END_VAR
IF PR_Load THEN PR_Load_Exe(); PR_Load:=FALSE; END_IF
IF PR_Save THEN PR_Save_Exe(); PR_Save:=FALSE; END_IF
IF CA_Load THEN CA_Load_Exe(); CA_Load:=FALSE; END_IF
IF CA_Save THEN CA_Save_Exe(); CA_Save:=FALSE; END_IF
IF JL_Load THEN JL_Load_Exe(); JL_Load:=FALSE; END_IF
IF JL_Save THEN JL_Save_Exe(); JL_Save:=FALSE; END_IF
END_FUNCTION_BLOCK
ACTION CA_Load_Exe:
sFileMode:='r';
FileOpen();

IF hFile<>0 THEN

	(* Read calendar month *)
	FOR i := 0 TO 31 DO
		r1:=SysFileSetPos(File:=hFile, Pos:=(1024 + ((CA_Sel-1)*32 + i)*4));
		r2:=SysFileRead(File:=hFile, Buffer:=ADR(CA.Profile[i]), Size:=1);
	END_FOR

	(* Close file *)
	SysFileClose(File:=hFile);

	(* Validate data *)
	CA_Act :=CA_Sel;
	CN_Act :=CN_Sel;
	CN_YAct:=CN_YSel;

	Message:='Calendar load OK';

END_IF
END_ACTION
ACTION CA_Save_Exe:
sFileMode:='a';
FileOpen();

IF hFile<>0 THEN

	(* Write calendar month *)
	FOR i := 0 TO 31 DO
		r1:=SysFileSetPos(File:=hFile, Pos:=(1024 + ((CA_Sel-1)*32 + i)*4));
		r2:=SysFileGetPos(hFile);
		r2:=SysFileWrite(File:=hFile, Buffer:=ADR(CA.Profile[i]), Size:=1);
	END_FOR

	(* Close file *)
	SysFileClose(File:=hFile);

	Message:='Calendar save OK';

END_IF
END_ACTION
ACTION FileOpen:
(* Create current filename 'yyyyCRnn.DAT' *)
sFileName:=CONCAT(FilesPath,WORD_TO_STRING(CN_YSel));
sFileName:=CONCAT(STR1:=sFileName, STR2:='CR');
IF CN_Sel<10 THEN
sFileName:=CONCAT(STR1:=sFileName, STR2:='0');
END_IF
sFileName:=CONCAT(STR1:=sFileName, STR2:=BYTE_TO_STRING(CN_Sel));
sFileName:=CONCAT(STR1:=sFileName, STR2:='.DAT');

(* Check file version and size! *)
(* ... *)

(* Open data file *)
hFile:=SysFileOpen(FileName:=sFileName, Mode:='r');

(* File not found *)
IF hFile=0 THEN
	Message:='File not found - created empty file';
	(* Create empty file *)
	hFile:=SysFileOpen(FileName:=sFileName, Mode:='w');
	MEMCLR(pDestinationAddress:=ADR(Buf), BytesToClear:=SIZEOF(Buf));
	FOR i := 0 TO 10239 BY 512 DO
		SysFileWrite(File:=hFile, Buffer:=ADR(Buf), Size:=512);
	END_FOR
	Buf[0]:=1;
	SysFileSetPos(File:=hFile, Pos:=0);
	SysFileWrite(File:=hFile, Buffer:=ADR(Buf), Size:=1);
END_IF

(* Close file *)
SysFileClose(File:=hFile);

(* Open data file *)
hFile:=SysFileOpen(FileName:=sFileName, Mode:=sFileMode);
END_ACTION
ACTION JL_Load_Exe:
sFileMode:='r';
FileOpen();

IF hFile<>0 THEN

	(* Read jolly *)
	r1:=SysFileSetPos(File:=hFile, Pos:=512);
	r2:=SysFileRead(File:=hFile, Buffer:=ADR(JL), Size:=SIZEOF(JL));

	(* Close file *)
	SysFileClose(File:=hFile);

	(* Validate data *)
	CN_Act:=CN_Sel;
	CN_YAct:=CN_YSel;

	Message:='Jolly load OK';

END_IF
END_ACTION
ACTION JL_Save_Exe:
sFileMode:='a';
FileOpen();

IF hFile<>0 THEN

	(* Write selected profile *)
	r1:=SysFileSetPos(File:=hFile, Pos:=512);
	r2:=SysFileWrite(File:=hFile, Buffer:=ADR(JL), Size:=SIZEOF(JL));

	(* Close file *)
	SysFileClose(File:=hFile);

	Message:='Jolly save OK';

END_IF
END_ACTION
ACTION PR_Load_Exe:
sFileMode:='r';
FileOpen();

IF hFile<>0 THEN

	(* Read selected profile *)
	r1:=SysFileSetPos(File:=hFile, Pos:=(3072 + 512*PR_Sel));
	r2:=SysFileRead(File:=hFile, Buffer:=ADR(PR), Size:=SIZEOF(PR));

	(* Close file *)
	SysFileClose(File:=hFile);

	(* Validate data *)
	PR_Act:=PR_Sel;
	CN_Act:=CN_Sel;
	CN_YAct:=CN_YSel;

	Message:='Profile load OK';

END_IF
END_ACTION
ACTION PR_Save_Exe:
sFileMode:='a';
FileOpen();

IF hFile<>0 THEN

	(* Write selected profile *)
	r1:=SysFileSetPos(File:=hFile, Pos:=(3072 + 512*PR_Sel));
	r2:=SysFileWrite(File:=hFile, Buffer:=ADR(PR), Size:=SIZEOF(PR));

	(* Close file *)
	SysFileClose(File:=hFile);

	Message:='Profile save OK';

END_IF
END_ACTION

(* POU Plant_Objects/obj_CRONTER, ST *)
FUNCTION_BLOCK obj_CRONTER
(* === THERMOSTAT ===
   v1.0[30/07/15] - Versioning
*)
VAR_INPUT
	(* Settings *)
	ID			: BYTE;		(* Index of instanced object *)

	InitOK		: BOOL;
	Alarm		: BOOL;
	Warning		: BOOL;

	Profile		: typ_Cron_Profile; 				(* Profilo attivo *)
	ProfileNr	: BYTE;								(* Indice profilo attivo *)
	CalendarIdx : WORD;								(* Indice calendario attivo *)
	Jolly		: ARRAY[0..9] OF typ_Cron_Jolly;	(* Jolly attivi *)

	Temperature	: INT;
	Local_MaxRunTAmb	:	INT;					(* Local maximum environment temperature, NOT "TAMB" *)

	Histeresys:INT; (* isteresi per la ripartenza del Comando ON*)
END_VAR
VAR_IN_OUT
END_VAR
VAR_OUTPUT
	SetPoint		: INT;
	Run				: BOOL;
	AntifreezeForce	: BOOL;
	RunCrono		: BOOL;

	(* Status *)
	Status_Log		: BYTE;
	Status_Vis 		: DWORD;
END_VAR
VAR
	Buf: 	ARRAY[0..512] OF BYTE; (* AVOID THIS!! *)
	hFile: 	DWORD;
	sFile: 	STRING;
	sFile2: STRING;

	i:		WORD;
	t1:		DWORD;
	t2:		BOOL;

END_VAR
(* Check initialization *)
IF NOT InitOK THEN Init(); END_IF

(* Check Temperature *)
(*IF Temperature < Local_MaxRunTAmb THEN*)

	(* LOCAL environment temperature lower than maximum allowed -> Proceed with SetPoint adjustment *)
	(* Chrono *)
	IF CalendarIdx<>Sys.Time_CT_Day THEN DB_Load(); END_IF
	SetPoint:=Profile.Setpoint[Sys.Time_CT_Quarter];

	(* Check jolly *)
	FOR i := 0 TO 9 DO
		IF ( DT_TO_DWORD(Jolly[i].Start)>0  AND Jolly[i].End>Jolly[i].Start AND
		     Jolly[i].Start<=Sys.Time_CT_DT AND Jolly[i].End>Sys.Time_CT_DT ) THEN
				SetPoint:=Jolly[i].Temp;
		END_IF
	END_FOR

(*
	IF SetPoint < 180 THEN
		(* Switch off the device *)
		Run := FALSE;
	ELSE
		(* Set according to feedback T - Histeresys of 1°C *)
		IF Temperature >= (SetPoint + 5) THEN
			Run := FALSE;
		ELSIF Temperature <= (SetPoint - 5) THEN
			Run := TRUE;
		END_IF

		(* Between "SetPoint-5" and "SetPoint+5" last state (ON or OFF) of "Run" is kept	*)
	END_IF
*)

(* Gestione uscita Crono *)
		IF SetPoint>0 THEN RunCrono := TRUE;
		ELSIF SetPoint=0 THEN RunCrono := FALSE;
		END_IF

(* GEstione uscita Cronotermostato *)


		IF Temperature >= (SetPoint) THEN
			Run := FALSE;
		ELSIF Temperature <= (SetPoint - Histeresys) THEN
			Run := TRUE;
		END_IF


(*ELSE
	(* Environment overtemperature: stop heating -> Stop device *)
	Run := FALSE;
END_IF
*)
(* Freeze warning: Switch on and heat! *)
(*IF Temperature < Plant_AntiFreezeTAmb THEN AntifreezeForce := TRUE;
ELSE AntifreezeForce := FALSE;
END_IF*)



(* Status color *)
   IF Alarm   THEN Status_Log:=2; Status_Vis:=COLOR_RED;
ELSIF Warning THEN Status_Log:=1; Status_Vis:=COLOR_YELLOW;
              ELSE Status_Log:=0; Status_Vis:=COLOR_GREEN;
			  END_IF
END_FUNCTION_BLOCK
ACTION AddLogData:
Logger.s1:=INSERT('&THER=',BYTE_TO_STRING(ID),5);
IF ID<10 THEN Logger.s1:=INSERT(Logger.s1,'0',5); END_IF

Logger.s1:=CONCAT(Logger.s1,INT_TO_STRING(SetPoint));			Logger.s1:=CONCAT(Logger.s1,';');

Logger.s1:=CONCAT(Logger.s1,WORD_TO_STRING(Status_Log));
ADDSTRING(ADR(Logger.TData), ADR(Logger.s1), Logger.TLen);
END_ACTION
ACTION DB_Create:
(* Create empty file *)
hFile:=SysFileOpen(FileName:=sFile, Mode:='w');

MEMCLR(pDestinationAddress:=ADR(Buf), BytesToClear:=SIZEOF(Buf));
FOR i := 0 TO 10239 BY 512 DO
	t1:=SysFileWrite(File:=hFile, Buffer:=ADR(Buf), Size:=512);		(* Clear created file (all bytes 0) *)
END_FOR
Buf[0]:=1;
t2:=SysFileSetPos(File:=hFile, Pos:=0);
t1:=SysFileWrite(File:=hFile, Buffer:=ADR(Buf), Size:=1);
SysFileClose(File:=hFile);
END_ACTION
ACTION DB_Load:
DB_SetName();

(* Open data file *)
hFile:=SysFileOpen(FileName:=sFile, Mode:='r');

(* File not found *)
IF hFile=0 THEN
	Warning:=TRUE;
	LogEv(EL_Wrn,EO_CRON,ID,1,'No_data_file');
	DB_Create();
	(* Reopen file *)
	hFile:=SysFileOpen(FileName:=sFile, Mode:='r');
	IF hfile=0 THEN
		Alarm:=TRUE;
		LogEv(EL_Alarm,EO_CRON,ID,3,'Filesystem_error');
		RETURN;
	END_IF
END_IF

(* Check version *)
SysFileRead(File:=hFile, Buffer:=ADR(Buf), Size:=1);
IF Buf[0]<>1 THEN
	IF NOT Alarm THEN
		Alarm:=TRUE;
		LogEv(EL_Alarm,EO_CRON,ID,2,'Bad_data_version');
	END_IF
	SysFileClose(File:=hFile);
	RETURN;
END_IF

(* Read Jolly data *)
t2:=SysFileSetPos(File:=hFile, Pos:=512);
t1:=SysFileRead(File:=hFile, Buffer:=ADR(Jolly), Size:=SIZEOF(Jolly));
(* Read active profile index *)
CalendarIdx:=Sys.Time_CT_Day;
t2:=SysFileSetPos(File:=hFile, Pos:=(1024+4*CalendarIdx));
t1:=SysFileRead(File:=hFile, Buffer:=ADR(ProfileNr), Size:=SIZEOF(ProfileNr));
(* Read active profile *)
t2:=SysFileSetPos(File:=hFile, Pos:=(3072+512*ProfileNr));
t1:=SysFileRead(File:=hFile, Buffer:=ADR(Profile), Size:=SIZEOF(Profile));

(* Close file and validate data *)
SysFileClose(File:=hFile);
END_ACTION
ACTION DB_SetName:
(* Create current filename 'yyyyCRnn.DAT' *)
sFile:=CONCAT(FilesPath,WORD_TO_STRING(Sys.Time_Year));
sFile:=CONCAT(STR1:=sFile, STR2:='CR');
IF ID<10 THEN
sFile:=CONCAT(STR1:=sFile, STR2:='0');
END_IF
sFile:=CONCAT(STR1:=sFile, STR2:=BYTE_TO_STRING(ID));
sFile:=CONCAT(STR1:=sFile, STR2:='.DAT');
END_ACTION
ACTION Init:
DB_Load();
InitOK:=TRUE;
END_ACTION

(* POU Plant_Objects/obj_MODBUS_ANZFRER_01, ST *)
FUNCTION_BLOCK obj_MODBUS_ANZFRER_01
VAR CONSTANT

	TimeOutModBus: TON;


END_VAR
VAR_INPUT
	ID			:	BYTE;
	Address		:	BYTE;
	(* Modbus *)
	Refresh_Now	:	BOOL;			(* Richiesta di lettura stato macchina Immediata  *)
	retryErrMax	:	BYTE := 2;

(*	IndirizzoDaScrivere: WORD;
	DatoDaScrivere: INT;
	ScriviDato: BOOL; *)

END_VAR
VAR_IN_OUT
	ModBus		:obj_MODBUS;

END_VAR
VAR_OUTPUT
	Status_Log	:	WORD;
	Status_Vis	:	DWORD;
END_VAR
VAR

	state		:	INT;
	retry		:	BYTE;
	retryErr	:	BYTE;
	ReadTmr		:	TON := (PT:=T#5s);
	fModbusAlr:BOOL;

(*	retry_write	:	BYTE;
	fWriteStatus:	BOOL;
	fWriteMode	:	BOOL;
	fWriteReset	:	BOOL; *)

	x: INT;

	VerificaFuctionCode: INT;
	VerificaNodoLetto: INT;
	ErroreComuModBus: BOOL;
	IndiceErrore: BYTE;

	MB_BitStato: ARRAY [0..450] OF BOOL;
	MB_RegistriLetti: ARRAY [0..450] OF INT;




	AddressRead: BYTE;
	index: BYTE;
	indexErr: BYTE;


	MB_V_L1_N: DWORD;
	MB_V_L2_N: DWORD;
	MB_V_L3_N: DWORD;
	MB_V_L1_L2: DWORD;
	MB_V_L1_L3: DWORD;
	MB_V_L2_L3: DWORD;
	MB_V_IL1: DWORD;
	MB_V_IL2: DWORD;
	MB_V_IL3: DWORD;
	MB_V_F: DWORD;
	MB_V_P: DWORD;
	MB_V_Q: DWORD;
	MB_V_P_F: DWORD;
	MB_IL1_MAX: DWORD;
	MB_IL2_MAX: DWORD;
	MB_IL3_MAX: DWORD;
	MB_PF_IL1: DWORD;
	MB_PF_IL2: DWORD;
	MB_PF_IL3: DWORD;
	MB_COSPI_IL1: DWORD;
	MB_COSPI_IL2: DWORD;
	MB_COSPI_IL3: DWORD;
	MB_V_P_AVG: DWORD;
	MB_V_P_MAX: DWORD;
	MB_V_Q_MAX: DWORD;
	MB_V_Q_AVG: DWORD;
	MB_V_KWh: DWORD;
	MB_V_kVAr: DWORD;



	moreno: ARRAY [0..20] OF WORD;
END_VAR
(* Call ModBus state machine *)
Stm();


(* Seganalzione stato Frigorifero  *)
IF ErroreComuModBus OR MB_BitStato[6] OR MB_BitStato[7] THEN
		Status_Log:=2; Status_Vis:=16#2020F0;
(*	ELSIF Warning OR Warning2 THEN
		Status_Log:=1; Status_Vis:=16#20F0F0; *)
    ELSE
		Status_Log:=0;
		Status_Vis:=16#006000;
END_IF
END_FUNCTION_BLOCK
ACTION AddLogData:
Logger.s1:=INSERT('&ANZ=',BYTE_TO_STRING(ID),4);
IF ID<10 THEN Logger.s1:=INSERT(Logger.s1,'0',4); END_IF


	Logger.s1:=CONCAT(Logger.s1,(REAL_TO_STRING(DWORD_TO_REAL(MB_V_L1_N)/1000)));
	Logger.s1:=CONCAT(Logger.s1,';');
	Logger.s1:=CONCAT(Logger.s1,(REAL_TO_STRING(DWORD_TO_REAL(MB_V_L2_N)/1000)));
	Logger.s1:=CONCAT(Logger.s1,';');
	Logger.s1:=CONCAT(Logger.s1,(REAL_TO_STRING(DWORD_TO_REAL(MB_V_L3_N)/1000)));
	Logger.s1:=CONCAT(Logger.s1,';');
	Logger.s1:=CONCAT(Logger.s1,(REAL_TO_STRING(DWORD_TO_REAL(MB_V_L1_L2)/1000)));
	Logger.s1:=CONCAT(Logger.s1,';');
	Logger.s1:=CONCAT(Logger.s1,(REAL_TO_STRING(DWORD_TO_REAL(MB_V_L1_L3)/1000)));
	Logger.s1:=CONCAT(Logger.s1,';');
	Logger.s1:=CONCAT(Logger.s1,(REAL_TO_STRING(DWORD_TO_REAL(MB_V_L2_L3)/1000)));
	Logger.s1:=CONCAT(Logger.s1,';');

	Logger.s1:=CONCAT(Logger.s1,(REAL_TO_STRING(DWORD_TO_REAL(MB_V_F))));
	Logger.s1:=CONCAT(Logger.s1,';');

	Logger.s1:=CONCAT(Logger.s1,(REAL_TO_STRING(DWORD_TO_REAL(MB_V_IL1))));
	Logger.s1:=CONCAT(Logger.s1,';');
	Logger.s1:=CONCAT(Logger.s1,(REAL_TO_STRING(DWORD_TO_REAL(MB_V_IL2))));
	Logger.s1:=CONCAT(Logger.s1,';');
	Logger.s1:=CONCAT(Logger.s1,(REAL_TO_STRING(DWORD_TO_REAL(MB_V_IL3))));
	Logger.s1:=CONCAT(Logger.s1,';');

	Logger.s1:=CONCAT(Logger.s1,(REAL_TO_STRING(DWORD_TO_REAL(MB_IL1_MAX))));
	Logger.s1:=CONCAT(Logger.s1,';');
	Logger.s1:=CONCAT(Logger.s1,(REAL_TO_STRING(DWORD_TO_REAL(MB_IL1_MAX))));
	Logger.s1:=CONCAT(Logger.s1,';');
	Logger.s1:=CONCAT(Logger.s1,(REAL_TO_STRING(DWORD_TO_REAL(MB_IL1_MAX))));
	Logger.s1:=CONCAT(Logger.s1,';');


	Logger.s1:=CONCAT(Logger.s1,(REAL_TO_STRING(DWORD_TO_REAL(MB_PF_IL1))));
	Logger.s1:=CONCAT(Logger.s1,';');
	Logger.s1:=CONCAT(Logger.s1,(REAL_TO_STRING(DWORD_TO_REAL(MB_PF_IL2))));
	Logger.s1:=CONCAT(Logger.s1,';');
	Logger.s1:=CONCAT(Logger.s1,(REAL_TO_STRING(DWORD_TO_REAL(MB_PF_IL3))));
	Logger.s1:=CONCAT(Logger.s1,';');

	Logger.s1:=CONCAT(Logger.s1,(REAL_TO_STRING(DWORD_TO_REAL(MB_V_P))));
	Logger.s1:=CONCAT(Logger.s1,';');
	Logger.s1:=CONCAT(Logger.s1,(REAL_TO_STRING(DWORD_TO_REAL(MB_V_P_AVG))));
	Logger.s1:=CONCAT(Logger.s1,';');
	Logger.s1:=CONCAT(Logger.s1,(REAL_TO_STRING(DWORD_TO_REAL(MB_V_P_MAX))));
	Logger.s1:=CONCAT(Logger.s1,';');

	Logger.s1:=CONCAT(Logger.s1,(REAL_TO_STRING(DWORD_TO_REAL(MB_V_Q))));
	Logger.s1:=CONCAT(Logger.s1,';');
	Logger.s1:=CONCAT(Logger.s1,(REAL_TO_STRING(DWORD_TO_REAL(MB_V_Q_MAX))));
	Logger.s1:=CONCAT(Logger.s1,';');

	Logger.s1:=CONCAT(Logger.s1,(REAL_TO_STRING(DWORD_TO_REAL(MB_V_KWh)/100)));
	Logger.s1:=CONCAT(Logger.s1,';');
	Logger.s1:=CONCAT(Logger.s1,(REAL_TO_STRING(DWORD_TO_REAL(MB_V_kVAr)/100)));
	Logger.s1:=CONCAT(Logger.s1,';');

	Logger.s1:=CONCAT(Logger.s1,WORD_TO_STRING(Status_Log));
	Logger.s1:=CONCAT(Logger.s1,';');

	Logger.s1:=CONCAT(Logger.s1,(REAL_TO_STRING(DWORD_TO_REAL(MB_COSPI_IL1))));
	Logger.s1:=CONCAT(Logger.s1,';');
	Logger.s1:=CONCAT(Logger.s1,(REAL_TO_STRING(DWORD_TO_REAL(MB_COSPI_IL2))));
	Logger.s1:=CONCAT(Logger.s1,';');
	Logger.s1:=CONCAT(Logger.s1,(REAL_TO_STRING(DWORD_TO_REAL(MB_COSPI_IL3))));
	Logger.s1:=CONCAT(Logger.s1,';');
	Logger.s1:=CONCAT(Logger.s1,'0');    (* 0=3-phase, 1 = mono phase *)


ADDSTRING(ADR(Logger.TData), ADR(Logger.s1), Logger.TLen);
END_ACTION
ACTION Stm:
CASE state OF
	0:	(* Refresh time manager *)
		ReadTmr(IN:=NOT ReadTmr.Q);
		(*A tempo interrogo il nodo sempre che non ci sia qualcuno che lo sta interrogando in quel momento *)

		IF (ReadTmr.Q AND NodoDaInterrogareANZ=Address )OR Refresh_Now AND NOT InibiscoModbusANZ THEN
			state := 10;
			ReadTmr.PT := T#5s;
			Refresh_Now := FALSE;
			InibiscoModbusANZ := TRUE;
		END_IF

	(**** Leggo le Analogiche a Disposzione  ****)

	10:	(* richiedo lettura Holding Registere Chiller  *)

		Modbus.MB_Query.SlaveAddress := Address;
		Modbus.MB_Query.FunctionCode := 3;
		ModBus.MB_Query.Read_StartAddress := 256 ;			(* richiedo lettura altri Parametri *)
		ModBus.MB_Query.Read_Quantity := 20;
		ModBus.MB_Start := TRUE;
		state := 20;

	20:	(* Risposta all'interrogazione *)
		IF NOT ModBus.MB_Start   THEN
			VerificaFuctionCode:=ModBus.MB_Resp.FunctionCode;
			VerificaNodoLetto:=ModBus.MB_Resp.SlaveAddress;

			IF ModBus.MB_MASTER.MB_Error<>0 THEN
				state := 300;
			ELSE
				MB_V_L1_N:= ModBus.MB_Resp.Data[0]*65536 +  ModBus.MB_Resp.Data[1];   	(* Vedi tabella *)
				MB_V_L2_N:= ModBus.MB_Resp.Data[2]*65536 +  ModBus.MB_Resp.Data[3];   	(* Vedi tabella *)
				MB_V_L3_N:= ModBus.MB_Resp.Data[4]*65536 +  ModBus.MB_Resp.Data[5];   	(* Vedi tabella *)
				MB_V_L1_L2:= ModBus.MB_Resp.Data[6]*65536 +  ModBus.MB_Resp.Data[7];   	(* Vedi tabella *)
				MB_V_L1_L3:= ModBus.MB_Resp.Data[8]*65536 +  ModBus.MB_Resp.Data[9];   	(* Vedi tabella *)
				MB_V_L2_L3:= ModBus.MB_Resp.Data[10]*65536 +  ModBus.MB_Resp.Data[11];   	(* Vedi tabella *)
				ModBus.MB_Query.Read_StartAddress := 268; 	(* richiedo lettura altri Parametri *)
				ModBus.MB_Query.Read_Quantity := 10;
				ModBus.MB_Start := TRUE;

				state := 30;
			END_IF
		END_IF

	30: (* Rispota Altri paramenti *)
		IF NOT ModBus.MB_Start  THEN

			IF ModBus.MB_MASTER.MB_Error<>0 THEN
				state := 300;
			ELSE
				MB_V_IL1:= ModBus.MB_Resp.Data[0]*65536 +  ModBus.MB_Resp.Data[1];   	(* Vedi tabella *)
				MB_V_IL2:= ModBus.MB_Resp.Data[2]*65536 +  ModBus.MB_Resp.Data[3];   	(* Vedi tabella *)
				MB_V_IL3:= ModBus.MB_Resp.Data[4]*65536 +  ModBus.MB_Resp.Data[5];   	(* Vedi tabella *)
				MB_V_F:= ModBus.MB_Resp.Data[6]*65536 +  ModBus.MB_Resp.Data[7];   	(* Vedi tabella *)
				MB_V_P:= ModBus.MB_Resp.Data[8]*65536 +  ModBus.MB_Resp.Data[9];   	(* Vedi tabella *)

				ModBus.MB_Query.Read_StartAddress := 278; (* richiedo lettura altri Parametri *)
				ModBus.MB_Query.Read_Quantity := 20;
				ModBus.MB_Start := TRUE;

				state := 40;
			END_IF
		END_IF



	40: (* Rispota Altri paramenti *)
		IF NOT ModBus.MB_Start  THEN

			IF ModBus.MB_MASTER.MB_Error<>0 THEN
				state := 300;
			ELSE
				MB_V_Q:= ModBus.MB_Resp.Data[0]*65536 +  ModBus.MB_Resp.Data[1];   	(* Vedi tabella *)
				MB_V_P_F:= ModBus.MB_Resp.Data[2]*65536 +  ModBus.MB_Resp.Data[3];   	(* Vedi tabella *)
				MB_V_KWh:= ModBus.MB_Resp.Data[4]*65536 +  ModBus.MB_Resp.Data[5];   	(* Vedi tabella *)
				MB_V_kVAr:= ModBus.MB_Resp.Data[6]*65536 +  ModBus.MB_Resp.Data[7];   	(* Vedi tabella *)

				ModBus.MB_Query.Read_StartAddress := 354; (* richiedo lettura altri Parametri *)
				ModBus.MB_Query.Read_Quantity := 20;
				ModBus.MB_Start := TRUE;

				state := 50;
			END_IF
		END_IF

	50: (* Rispota Altri paramenti *)
		IF NOT ModBus.MB_Start  THEN

			IF ModBus.MB_MASTER.MB_Error<>0 THEN
				state := 300;
			ELSE

				MB_V_P_AVG:= ModBus.MB_Resp.Data[0]*65536 +  ModBus.MB_Resp.Data[1];   	(* Vedi tabella *)
				MB_V_P_MAX:= ModBus.MB_Resp.Data[2]*65536 +  ModBus.MB_Resp.Data[3];   	(* Vedi tabella *)
				MB_IL1_MAX:= ModBus.MB_Resp.Data[4]*65536 +  ModBus.MB_Resp.Data[5];   	(* Vedi tabella *)
				MB_IL2_MAX:= ModBus.MB_Resp.Data[6]*65536 +  ModBus.MB_Resp.Data[7];   	(* Vedi tabella *)
				MB_IL3_MAX:= ModBus.MB_Resp.Data[8]*65536 +  ModBus.MB_Resp.Data[9];   	(* Vedi tabella *)

				ModBus.MB_Query.Read_StartAddress := 342; (* richiedo lettura altri Parametri *)
				ModBus.MB_Query.Read_Quantity := 20;
				ModBus.MB_Start := TRUE;

				state := 55;
			END_IF
		END_IF

	55: (* Rispota Altri paramenti *)
		IF NOT ModBus.MB_Start  THEN

			IF ModBus.MB_MASTER.MB_Error<>0 THEN
				state := 300;
			ELSE
				MB_PF_IL1:= ModBus.MB_Resp.Data[0]*65536 +  ModBus.MB_Resp.Data[1];   	(* Vedi tabella *)
				MB_PF_IL2:= ModBus.MB_Resp.Data[2]*65536 +  ModBus.MB_Resp.Data[3];   	(* Vedi tabella *)
				MB_PF_IL3:= ModBus.MB_Resp.Data[4]*65536 +  ModBus.MB_Resp.Data[5];   	(* Vedi tabella *)
				MB_COSPI_IL1:= ModBus.MB_Resp.Data[6]*65536 +  ModBus.MB_Resp.Data[7];   	(* Vedi tabella *)
				MB_COSPI_IL2:= ModBus.MB_Resp.Data[8]*65536 +  ModBus.MB_Resp.Data[9];   	(* Vedi tabella *)
				MB_COSPI_IL3:= ModBus.MB_Resp.Data[10]*65536 +  ModBus.MB_Resp.Data[11];   	(* Vedi tabella *)

				ModBus.MB_Query.Read_StartAddress := 422; (* richiedo lettura altri Parametri *)
				ModBus.MB_Query.Read_Quantity := 20;
				ModBus.MB_Start := TRUE;

				state := 60;
			END_IF
		END_IF

	60: (* Rispota Altri paramenti *)
		IF NOT ModBus.MB_Start  THEN

			IF ModBus.MB_MASTER.MB_Error<>0 THEN
				state := 300;
			ELSE
				MB_V_Q_MAX:= ModBus.MB_Resp.Data[0]*65536 +  ModBus.MB_Resp.Data[1];   	(* Vedi tabella *)
				MB_V_Q_AVG:= ModBus.MB_Resp.Data[2]*65536 +  ModBus.MB_Resp.Data[3];   	(* Vedi tabella *)

				(* ModBus.MB_Query.Read_StartAddress := 422; (* richiedo lettura altri Parametri *)
				ModBus.MB_Query.Read_Quantity := 20;
				ModBus.MB_Start := TRUE; *)

				state := 295;
			END_IF
		END_IF





		295:
		IF NOT ModBus.MB_Start THEN
			IF ModBus.MB_MASTER.MB_Error<>0 THEN (*OR ModBus.MB_MASTER.MB_Error<>0 THEN*)
				state := 300;
			ELSE
				IF fModbusAlr THEN fModbusAlr := FALSE; END_IF
				NodoDaInterrogareANZ:=Address+1;
				InibiscoModbusANZ:=FALSE;
				retryErr := 0;
				retry := 0;
				state := 0;
					IF fModbusAlr=FALSE AND ErroreComuModBus=TRUE THEN
						LogEv(EL_Log,EO_CHI,ID,62,'ComunicazioneModBus_OK');
						ErroreComuModBus := FALSE;
				(*	WarningCtr := SEL(WarningCtr=0, WarningCtr-1, 0); *)
					END_IF


			END_IF
		END_IF



	(**** CHECK MODBUS ERROR ****)
	300: 	(* Release MODBUS *)
			InibiscoModbusANZ:=FALSE;
			(* Retries *)
			retry:=retry+1;
			IF retry>3 THEN
				retry:=0;

				(* Verify if slave is dead *)
				IF retryErr < retryErrMaX THEN
					retryErr := retryErr + 1;
				ELSE
					fModbusAlr := TRUE;
					(* Verify ModBus error	*)

					IF fModbusAlr AND ErroreComuModBus=FALSE THEN
						LogEv(EL_Alarm,EO_CHI,ID,61,CONCAT('ErroreModbus_',INT_TO_STRING(ModBus.MB_MASTER.MB_Error)));
						ErroreComuModBus := TRUE;
					END_IF
				END_IF

				END_IF
			Refresh_Now := FALSE;
			InibiscoModbusANZ:=FALSE;
			NodoDaInterrogareANZ:=Address+1;
			state:=0;
END_CASE




(* Controllo Time Out Ciclo ModBus *)

TimeOutModBus(In:=state<>0,PT:=t#30s);
IF TimeOutModBus.Q THEN
	State:=0;
	Refresh_Now:=TRUE;  (* Rilancio la lettura del nodo *)
	IF MODBUS.MB_Lock=TRUE THEN MODBUS.MB_Lock:=FALSE;END_IF
	IF InibiscoModbusANZ=TRUE THEN InibiscoModbusANZ:=FALSE;END_IF
END_IF
END_ACTION

(* POU Plant_Objects/obj_MODBUS_FRG_AER485P1, ST *)
FUNCTION_BLOCK obj_MODBUS_FRG_AER485P1
VAR CONSTANT

	TimeOutModBus: TON;


END_VAR
VAR_INPUT
	ID			:	BYTE;
	Address		:	BYTE;


	SetPointManuale: INT; 			(* SetPoint forazato in manuale escludendo la curva di carico *)
	AbilitaSetPointManuale : BOOL ; (* Abilita il funzionamento col set point Manaule Escludendo la curva cliamtica *)


	(* Modbus *)
	Refresh_Now	:	BOOL;			(* Richiesta di lettura stato macchina Immediata  *)
	retryErrMax	:	BYTE := 2;

	Temperatura: INT;


	STOP_REQ: BOOL;
	RUN_REQ: BOOL;
	(* Timings *)
	OnDelay		:	TIME;
	OffDelay	:	TIME;

	OnOff		: 	BOOL;

	IndirizzoDaScrivere: WORD;
	DatoDaScrivere: INT;
	ScriviDato: BOOL;

	ImpMB_2SetPoint: INT;
	ImpMB_ResetFrigo: BOOL;
	ImpMB_LocRem: BOOL;
	fWriteAttivazioneComandi:BOOL;




END_VAR
VAR_IN_OUT
	ModBus		:obj_MODBUS;
	CLIM		:typ_Clima;

END_VAR
VAR_OUTPUT
	Run			:	BOOL;

	Status_Log	:	WORD;
	Status_Vis	:	DWORD;
END_VAR
VAR
	(* da diego per gestione stato stringa > 255*)
	temp :STRING(255);
	tempRaw		: ARRAY [0..MAX_SEND_TCP_CLIENT] OF BYTE;
	tempRawLen :DINT;
	longString:STRING(800);

	(* Timer manage switch on/off delay *)
	Delay		: 	TONOF;

	AllarmeFrigo_MB		:ARRAY [0..100] OF	FLT_EVENT;
	Warning		:	FLT_TAP := (TAP:=100);

	state		:	INT;
	retry		:	BYTE;
	retryErr	:	BYTE;
	ReadTmr		:	TON := (PT:=T#5s);
	fModbusAlr:BOOL;

(*	retry_write	:	BYTE;
	fWriteStatus:	BOOL;
	fWriteMode	:	BOOL;
	fWriteReset	:	BOOL; *)

	SetPointCC: DINT;
	x: INT;
	ImpMB_SetPoint: INT;
	Ctrl_Run: BOOL;


	VerificaFuctionCode: INT;
	VerificaNodoLetto: INT;
	ErroreComuModBus: BOOL;
	IndiceErrore: BYTE;

	MB_BitStato: ARRAY [0..200] OF BOOL;
	MB_RegistriLetti: ARRAY [0..450] OF INT;


	AddressRead: BYTE;
	index: BYTE;
	indexErr: BYTE;





END_VAR
VAR_INPUT RETAIN
	ChillerAbilitato: BOOL;
END_VAR
(* Aggiornamento in tempo reale dei TON e TOFF funzionamento Pompa *)

Delay.PT_OF := OffDelay;
Delay.PT_ON := OnDelay + WORD_TO_TIME(1000*ID);

(* Check climatic setup *)
IF NOT CLIM.InitOK THEN Clima_Default(); END_IF;
(* Calculate Setpoint *)

	IF Temperatura>=CLIM.Points[0].X  THEN SetPointCC:=CLIM.Points[0].Y; END_IF;
	IF Temperatura>=CLIM.Points[1].X AND Temperatura<CLIM.Points[0].X THEN SetPointCC:=CLIM.Points[0].Y; END_IF;
	IF Temperatura>=CLIM.Points[2].X AND Temperatura<CLIM.Points[1].X THEN SetPointCC:=CLIM.Points[1].Y; END_IF;
	IF Temperatura>=CLIM.Points[3].X AND Temperatura<CLIM.Points[2].X THEN SetPointCC:=CLIM.Points[2].Y; END_IF;
	IF Temperatura>=CLIM.Points[4].X AND Temperatura<CLIM.Points[3].X THEN SetPointCC:=CLIM.Points[3].Y; END_IF;
	IF Temperatura<CLIM.Points[4].X THEN SetPointCC:=CLIM.Points[4].Y; END_IF;


	IF Temperatura<CLIM.Points[4].X THEN SetPointCC:=CLIM.Points[4].Y; END_IF;


(* Scelta del set point della cladaia o vien preso dalla curva cliamtica o da un riferimento esterno *)
IF AbilitaSetPointManuale THEN
	ImpMB_SetPoint:=(SetPointManuale);
ELSE
	ImpMB_SetPoint:=DINT_TO_INT(SetPointCC);
END_IF


(* Controllo Bit di funzionamento ON e OFF  *)
Ctrl_Run := OnOff AND ChillerAbilitato;
Delay(IN:=Ctrl_Run);



IF STOP_REQ THEN Run := 1;
	ELSIF RUN_REQ THEN Run := 0;
ELSE
	Run :=Delay.OUT AND ChillerAbilitato;
END_IF



(* Call ModBus state machine *)
Stm();

(* Check alarm	*)
CheckAlarm();



(* Seganalzione stato Frigorifero  *)
IF ErroreComuModBus OR MB_BitStato[6] OR MB_BitStato[7] THEN
		Status_Log:=2; Status_Vis:=16#2020F0;
(*	ELSIF Warning OR Warning2 THEN
		Status_Log:=1; Status_Vis:=16#20F0F0; *)
    ELSE
		Status_Log:=0;
		Status_Vis:=16#006000;
END_IF
END_FUNCTION_BLOCK
ACTION AddLogData:
Logger.s1:=INSERT('&CHI=',BYTE_TO_STRING(ID),4);
IF ID<10 THEN Logger.s1:=INSERT(Logger.s1,'0',4); END_IF

tempRawLen:=0;

temp:=Logger.s1;
ADDSTRING(ADR(tempRaw), ADR(temp), tempRawLen);

FOR x:= 1 TO 2 DO

	temp:=CONCAT(INT_TO_STRING(MB_RegistriLetti[x]),';');
	ADDSTRING(ADR(tempRaw), ADR(temp), tempRawLen);

END_FOR


FOR x:= 5 TO 15 DO
	temp:=CONCAT(INT_TO_STRING(MB_RegistriLetti[x]),';');
	ADDSTRING(ADR(tempRaw), ADR(temp), tempRawLen);
END_FOR

FOR x:= 18 TO 19 DO
	temp:=CONCAT(INT_TO_STRING(MB_RegistriLetti[x]),';');
	ADDSTRING(ADR(tempRaw), ADR(temp), tempRawLen);
END_FOR

FOR x:= 21 TO 25 DO
	temp:=CONCAT(INT_TO_STRING(MB_RegistriLetti[x]),';');
	ADDSTRING(ADR(tempRaw), ADR(temp), tempRawLen);
END_FOR

FOR x:= 180 TO 207 DO
	temp:=CONCAT(INT_TO_STRING(MB_RegistriLetti[x]),';');
	ADDSTRING(ADR(tempRaw), ADR(temp), tempRawLen);
END_FOR

FOR x:= 209 TO 232 DO
		temp:=CONCAT(INT_TO_STRING(MB_RegistriLetti[x]),';');
	ADDSTRING(ADR(tempRaw), ADR(temp), tempRawLen);
END_FOR

FOR x:= 235 TO 244 DO
	temp:=CONCAT(INT_TO_STRING(MB_RegistriLetti[x]),';');
	ADDSTRING(ADR(tempRaw), ADR(temp), tempRawLen);
END_FOR

FOR x:= 268 TO 276 DO
	temp:=CONCAT(INT_TO_STRING(MB_RegistriLetti[x]),';');
	ADDSTRING(ADR(tempRaw), ADR(temp), tempRawLen);
END_FOR

FOR x:= 408 TO 414 DO
	temp:=CONCAT(INT_TO_STRING(MB_RegistriLetti[x]),';');
	ADDSTRING(ADR(tempRaw), ADR(temp), tempRawLen);
END_FOR

FOR x:= 1 TO 19 DO
	temp:=CONCAT(SEL(MB_BitStato[x],'0','1'),';');
	ADDSTRING(ADR(tempRaw), ADR(temp), tempRawLen);
END_FOR

FOR x:= 21 TO 21 DO
	temp:=CONCAT(SEL(MB_BitStato[x],'0','1'),';');
	ADDSTRING(ADR(tempRaw), ADR(temp), tempRawLen);
END_FOR

FOR x:= 28 TO 31 DO
	temp:=CONCAT(SEL(MB_BitStato[x],'0','1'),';');
	ADDSTRING(ADR(tempRaw), ADR(temp), tempRawLen);
END_FOR

FOR x:= 34 TO 59 DO
	temp:=CONCAT(SEL(MB_BitStato[x],'0','1'),';');
	ADDSTRING(ADR(tempRaw), ADR(temp), tempRawLen);
END_FOR

FOR x:= 100 TO 198 DO
	temp:=CONCAT(SEL(MB_BitStato[x],'0','1'),';');
	ADDSTRING(ADR(tempRaw), ADR(temp), tempRawLen);
END_FOR

temp:=SEL(MB_BitStato[199],'0','1');
ADDSTRING(ADR(tempRaw), ADR(temp), tempRawLen);



(*



Logger.s1:=CONCAT(Logger.s1,(INT_TO_STRING(MB_RegistriLetti[204])); 			(* Set modo funzionamento freddo *)
Logger.s1:=CONCAT(Logger.s1,';');
Logger.s1:=CONCAT(Logger.s1,(INT_TO_STRING(MB_RegistriLetti[206]));  			(* SetCaldo Set modo funzionamento caldo *)
Logger.s1:=CONCAT(Logger.s1,';');
Logger.s1:=CONCAT(Logger.s1,WORD_TO_STRING(MB_DifGradi));  			(* Dif.Grad Set differenziale gradino per termostato *)
Logger.s1:=CONCAT(Logger.s1,';');
Logger.s1:=CONCAT(Logger.s1,WORD_TO_STRING(MB_DifTot));    			(* Dif.Tot. Set differenziale totale per termostato *)
Logger.s1:=CONCAT(Logger.s1,';');
Logger.s1:=CONCAT(Logger.s1,WORD_TO_STRING(MB_Temp_InH2O)); 		(* Temperatura ingresso acqua *)
Logger.s1:=CONCAT(Logger.s1,';');
Logger.s1:=CONCAT(Logger.s1,WORD_TO_STRING(MB_TUA_C1));				(* Temperatura uscita acqua circuito 1 *)
Logger.s1:=CONCAT(Logger.s1,';');
Logger.s1:=CONCAT(Logger.s1,WORD_TO_STRING(MB_SecondoSetFreddo));	(* Secondo set freddo *)
Logger.s1:=CONCAT(Logger.s1,';');
Logger.s1:=CONCAT(Logger.s1,WORD_TO_STRING(MB_h_CP1));				(*Ore funzionamento compressore circuito 1 *)
Logger.s1:=CONCAT(Logger.s1,';');
Logger.s1:=CONCAT(Logger.s1,WORD_TO_STRING(MB_h_CP2));				(* Ore funzionamento compressore circuito 2 *)
Logger.s1:=CONCAT(Logger.s1,';');
Logger.s1:=CONCAT(Logger.s1,WORD_TO_STRING(MB_h_CP1A));				(* Ore funzionamento compressore circuito 2 *)
Logger.s1:=CONCAT(Logger.s1,';');

Logger.s1:=CONCAT(Logger.s1,WORD_TO_STRING(Status_Log));
Logger.s1:=CONCAT(Logger.s1,';');
Logger.s1:=CONCAT(Logger.s1,SEL(ChillerAbilitato,'0','1')); (* Chiller Abilitato 0=Disabilitato   1=abilitato *)
Logger.s1:=CONCAT(Logger.s1,';');
Logger.s1:=CONCAT(Logger.s1,SEL(MB_BitStato[0],'0','1')); 	(* Comando standby/acceso (toggle)0=OFF   1=ON *)
Logger.s1:=CONCAT(Logger.s1,';');
Logger.s1:=CONCAT(Logger.s1,SEL(MB_BitStato[1],'0','1'));	(* Comando modo funzionamento freddo/caldo (toggle) 0=FREDDO 1=CALDO *)
Logger.s1:=CONCAT(Logger.s1,';');
Logger.s1:=CONCAT(Logger.s1,SEL(MB_BitStato[2],'0','1'));	(* Comando reset sicurezze1=RESET  *)
Logger.s1:=CONCAT(Logger.s1,';');
Logger.s1:=CONCAT(Logger.s1,SEL(MB_BitStato[3],'0','1'));	 (* Comando locale/remoto (toggle)0=LOCALE   1=REMOTO  *)
Logger.s1:=CONCAT(Logger.s1,';');
Logger.s1:=CONCAT(Logger.s1,SEL(MB_BitStato[6],'0','1'));	(* Stato riassunto allarmi circuito 1  *)
Logger.s1:=CONCAT(Logger.s1,';');
Logger.s1:=CONCAT(Logger.s1,SEL(MB_BitStato[7],'0','1'));	(* Stato riassunto allarmi circuito 2  *)
Logger.s1:=CONCAT(Logger.s1,';');
Logger.s1:=CONCAT(Logger.s1,SEL(MB_BitStato[8],'0','1'));	(* Allarme flussostato *)
Logger.s1:=CONCAT(Logger.s1,';');
Logger.s1:=CONCAT(Logger.s1,SEL(MB_BitStato[12],'0','1'));	(*  Allarme termica compressore circuito 1  *)
Logger.s1:=CONCAT(Logger.s1,';');
Logger.s1:=CONCAT(Logger.s1,SEL(MB_BitStato[13],'0','1'));	(*  Allarme bassa pressione circuito 1   *)
Logger.s1:=CONCAT(Logger.s1,';');
Logger.s1:=CONCAT(Logger.s1,SEL(MB_BitStato[14],'0','1'));	(*  Allarme alta pressione circuito 1   *)
Logger.s1:=CONCAT(Logger.s1,';');
Logger.s1:=CONCAT(Logger.s1,SEL(MB_BitStato[15],'0','1'));	(*   Allarme antigelo circuito 1   *)
Logger.s1:=CONCAT(Logger.s1,';');
Logger.s1:=CONCAT(Logger.s1,SEL(MB_BitStato[16],'0','1'));	(*    Allarme termica ventilatore circuito 1   *)
Logger.s1:=CONCAT(Logger.s1,';');
Logger.s1:=CONCAT(Logger.s1,SEL(MB_BitStato[19],'0','1'));	(*  Allarme termica compressore circuito 2  *)
Logger.s1:=CONCAT(Logger.s1,';');
Logger.s1:=CONCAT(Logger.s1,SEL(MB_BitStato[20],'0','1'));  (*  Allarme bassa pressione circuito 2   *)
Logger.s1:=CONCAT(Logger.s1,';');
Logger.s1:=CONCAT(Logger.s1,SEL(MB_BitStato[21],'0','1'));  (*  Allarme alta pressione circuito 2   *)
Logger.s1:=CONCAT(Logger.s1,';');
Logger.s1:=CONCAT(Logger.s1,SEL(MB_BitStato[22],'0','1'));  (*   Allarme antigelo circuito 2   *)
Logger.s1:=CONCAT(Logger.s1,';');
Logger.s1:=CONCAT(Logger.s1,SEL(MB_BitStato[23],'0','1'));  (*    Allarme termica ventilatore circuito 2   *)
Logger.s1:=CONCAT(Logger.s1,';');
Logger.s1:=CONCAT(Logger.s1,SEL(MB_BitStato[26],'0','1'));  (*    Allarme monitore di tensione   *)
Logger.s1:=CONCAT(Logger.s1,';');
Logger.s1:=CONCAT(Logger.s1,SEL(MB_BitStato[29],'0','1'));  (*    Allarme Eprom   *)
Logger.s1:=CONCAT(Logger.s1,';');
Logger.s1:=CONCAT(Logger.s1,SEL(MB_BitStato[31],'0','1'));  (*     Carico pompa evaporatore   *)
Logger.s1:=CONCAT(Logger.s1,';');
Logger.s1:=CONCAT(Logger.s1,SEL(MB_BitStato[34],'0','1'));  (*      Carico compressore circuito 1   *)
Logger.s1:=CONCAT(Logger.s1,';');
Logger.s1:=CONCAT(Logger.s1,SEL(MB_BitStato[38],'0','1'));  (*       Carico ventilatore circuito 1   *)
Logger.s1:=CONCAT(Logger.s1,';');
Logger.s1:=CONCAT(Logger.s1,SEL(MB_BitStato[40],'0','1'));  (*        Carico valvola liquido circuito 1   *)
Logger.s1:=CONCAT(Logger.s1,';');
Logger.s1:=CONCAT(Logger.s1,SEL(MB_BitStato[41],'0','1'));  (*         Carico compressore secondario circuito 1   *)
Logger.s1:=CONCAT(Logger.s1,';');
Logger.s1:=CONCAT(Logger.s1,SEL(MB_BitStato[42],'0','1'));  (*         Carico compressore circuito 2   *)
Logger.s1:=CONCAT(Logger.s1,';');
Logger.s1:=CONCAT(Logger.s1,SEL(MB_BitStato[46],'0','1'));  (*         Carico ventilatore circuito 2    *)
Logger.s1:=CONCAT(Logger.s1,';');
Logger.s1:=CONCAT(Logger.s1,SEL(MB_BitStato[48],'0','1'));  (*          Carico valvola liquido circuito 2    *)
Logger.s1:=CONCAT(Logger.s1,';');
Logger.s1:=CONCAT(Logger.s1,SEL(MB_BitStato[81],'0','1'));  (*           Allarme termica compressore circuito 1A     *)
Logger.s1:=CONCAT(Logger.s1,';');
Logger.s1:=CONCAT(Logger.s1,SEL(MB_BitStato[86],'0','1'));  (*          Allarme antigelo evaporatore circuito 1     *)
Logger.s1:=CONCAT(Logger.s1,';');
Logger.s1:=CONCAT(Logger.s1,SEL(MB_BitStato[87],'0','1'));  (*          Allarme antigelo evaporatore circuito 2     *)




*)


ADDSTRING(ADR(Logger.TData), ADR(tempRaw), Logger.TLen);
END_ACTION
ACTION CheckAlarm:
(**** GEstione Log ad Evento *****)


FOR x:=0 TO 100 DO

	AllarmeFrigo_MB[x](IN:=MB_BitStato[x+100] );

	IF AllarmeFrigo_MB[x].EVH THEN
		LogEv(EL_Log,EO_CHI,ID,x+100,CONCAT ('Allarme Attivo n. ', INT_TO_STRING(x+100)));
	END_IF

	IF AllarmeFrigo_MB[x].EVL THEN
		LogEv(EL_Log,EO_CHI,ID,x+100,CONCAT ('Allarme Rientrato n. ', INT_TO_STRING(x+100)));
	END_IF

END_FOR
END_ACTION
ACTION Clima_Default:
IF CLIM.Points[0].X=0 THEN
	CLIM.Points[0].X:=-300; CLIM.Points[0].Y:=770;
	CLIM.Points[1].X:=-70 ; CLIM.Points[1].Y:=770;
	CLIM.Points[2].X:= 80; 	CLIM.Points[2].Y:=690;
	CLIM.Points[3].X:= 200; CLIM.Points[3].Y:=300;
	CLIM.Points[4].X:= 500; CLIM.Points[4].Y:=200;
END_IF
CLIM.InitOK:=TRUE;
LogEv(EL_Wrn,EO_chi,ID,0,'Climatic_default');
END_ACTION
ACTION Stm:
CASE state OF
	0:	(* Refresh time manager *)
		ReadTmr(IN:=NOT ReadTmr.Q);
		(*A tempo interrogo il nodo sempre che non ci sia qualcuno che lo sta interrogando in quel momento *)

		IF (ReadTmr.Q AND NodoDaInterrogareChiller=Address )OR Refresh_Now AND NOT InibiscoModbusChiller THEN
			state := 10;
			ReadTmr.PT := T#5s;  (* moreno *)
			Refresh_Now := FALSE;
			InibiscoModbusChiller := TRUE;
		END_IF

	(**** Leggo le Analogiche a Disposzione  ****)

	10:	(* richiedo lettura Holding Registere Chiller  *)

		Modbus.MB_Query.SlaveAddress := Address;
		Modbus.MB_Query.FunctionCode := 3;
		ModBus.MB_Query.Read_StartAddress := 0 ;			(* richiedo lettura altri Parametri *)
		ModBus.MB_Query.Read_Quantity := 3;
		ModBus.MB_Start := TRUE;
		state := 20;

	20:	(* Risposta all'interrogazione *)
		IF NOT ModBus.MB_Start   THEN
			VerificaFuctionCode:=ModBus.MB_Resp.FunctionCode;
			VerificaNodoLetto:=ModBus.MB_Resp.SlaveAddress;

			IF ModBus.MB_MASTER.MB_Error<>0 THEN
				state := 300;
			ELSE
				MB_RegistriLetti[0] := ModBus.MB_Resp.Data[0];   	(* Vedi tabella *)
				MB_RegistriLetti[1] := ModBus.MB_Resp.Data[1];		(* Vedi tabella *)
				MB_RegistriLetti[2] := ModBus.MB_Resp.Data[2];		(* Vedi tabella *)


				ModBus.MB_Query.Read_StartAddress := 5; 	(* richiedo lettura altri Parametri *)
				ModBus.MB_Query.Read_Quantity := 11;
				ModBus.MB_Start := TRUE;

				state := 30;
			END_IF
		END_IF

	30: (* Rispota Altri paramenti *)
		IF NOT ModBus.MB_Start  THEN

			IF ModBus.MB_MASTER.MB_Error<>0 THEN
				state := 300;
			ELSE
				MB_RegistriLetti[5] := ModBus.MB_Resp.Data[0];   	(* Vedi tabella *)
				MB_RegistriLetti[6] := ModBus.MB_Resp.Data[1];		(* Vedi tabella *)
				MB_RegistriLetti[7] := ModBus.MB_Resp.Data[2];		(* Vedi tabella *)
				MB_RegistriLetti[8] := ModBus.MB_Resp.Data[3];		(* Vedi tabella *)
				MB_RegistriLetti[9] := ModBus.MB_Resp.Data[4];		(* Vedi tabella *)
				MB_RegistriLetti[10] := ModBus.MB_Resp.Data[5];		(* Vedi tabella *)
				MB_RegistriLetti[11] := ModBus.MB_Resp.Data[6];		(* Vedi tabella *)
				MB_RegistriLetti[12] := ModBus.MB_Resp.Data[7];		(* Vedi tabella *)
				MB_RegistriLetti[13] := ModBus.MB_Resp.Data[8];		(* Vedi tabella *)
				MB_RegistriLetti[14] := ModBus.MB_Resp.Data[9];		(* Vedi tabella *)
				MB_RegistriLetti[15] := ModBus.MB_Resp.Data[10];		(* Vedi tabella *)

				ModBus.MB_Query.Read_StartAddress := 21; (* richiedo lettura altri Parametri *)
				ModBus.MB_Query.Read_Quantity := 5;
				ModBus.MB_Start := TRUE;

				state := 40;
			END_IF
		END_IF

	40: (* Rispota Altri paramenti *)
		IF NOT ModBus.MB_Start  THEN

			IF ModBus.MB_MASTER.MB_Error<>0 THEN
				state := 300;
			ELSE
				MB_RegistriLetti[21] := ModBus.MB_Resp.Data[0];   	(* Vedi tabella *)
				MB_RegistriLetti[22] := ModBus.MB_Resp.Data[1];		(* Vedi tabella *)
				MB_RegistriLetti[23] := ModBus.MB_Resp.Data[2];		(* Vedi tabella *)
				MB_RegistriLetti[24] := ModBus.MB_Resp.Data[3];		(* Vedi tabella *)
				MB_RegistriLetti[25] := ModBus.MB_Resp.Data[4];		(* Vedi tabella *)

				ModBus.MB_Query.Read_StartAddress := 180; (* richiedo lettura altri Parametri *)
				ModBus.MB_Query.Read_Quantity := 20;
				ModBus.MB_Start := TRUE;

				state := 45;
			END_IF
		END_IF

	45: (* Rispota Altri paramenti *)
		IF NOT ModBus.MB_Start  THEN

			IF ModBus.MB_MASTER.MB_Error<>0 THEN
				state := 300;
			ELSE
				MB_RegistriLetti[180] := ModBus.MB_Resp.Data[0];   	(* Vedi tabella *)
				MB_RegistriLetti[181] := ModBus.MB_Resp.Data[1];		(* Vedi tabella *)
				MB_RegistriLetti[182] := ModBus.MB_Resp.Data[2];		(* Vedi tabella *)
				MB_RegistriLetti[183] := ModBus.MB_Resp.Data[3];		(* Vedi tabella *)
				MB_RegistriLetti[184] := ModBus.MB_Resp.Data[4];		(* Vedi tabella *)
				MB_RegistriLetti[185] := ModBus.MB_Resp.Data[5];		(* Vedi tabella *)
				MB_RegistriLetti[186] := ModBus.MB_Resp.Data[6];		(* Vedi tabella *)
				MB_RegistriLetti[187] := ModBus.MB_Resp.Data[7];		(* Vedi tabella *)
				MB_RegistriLetti[188] := ModBus.MB_Resp.Data[8];		(* Vedi tabella *)
				MB_RegistriLetti[189] := ModBus.MB_Resp.Data[9];		(* Vedi tabella *)
				MB_RegistriLetti[190] := ModBus.MB_Resp.Data[10];		(* Vedi tabella *)
				MB_RegistriLetti[191] := ModBus.MB_Resp.Data[11];		(* Vedi tabella *)
				MB_RegistriLetti[192] := ModBus.MB_Resp.Data[12];		(* Vedi tabella *)
				MB_RegistriLetti[193] := ModBus.MB_Resp.Data[13];		(* Vedi tabella *)
				MB_RegistriLetti[194] := ModBus.MB_Resp.Data[14];		(* Vedi tabella *)
				MB_RegistriLetti[195] := ModBus.MB_Resp.Data[15];		(* Vedi tabella *)
				MB_RegistriLetti[196] := ModBus.MB_Resp.Data[16];		(* Vedi tabella *)
				MB_RegistriLetti[197] := ModBus.MB_Resp.Data[17];		(* Vedi tabella *)
				MB_RegistriLetti[198] := ModBus.MB_Resp.Data[18];		(* Vedi tabella *)
				MB_RegistriLetti[199] := ModBus.MB_Resp.Data[19];		(* Vedi tabella *)

				ModBus.MB_Query.Read_StartAddress := 200; (* richiedo lettura altri Parametri *)
				ModBus.MB_Query.Read_Quantity := 9;
				ModBus.MB_Start := TRUE;

				state := 50;
			END_IF
		END_IF
	50: (* Rispota Altri paramenti *)
		IF NOT ModBus.MB_Start  THEN

			IF ModBus.MB_MASTER.MB_Error<>0 THEN
				state := 300;
			ELSE
				MB_RegistriLetti[200] := ModBus.MB_Resp.Data[0];   	(* Vedi tabella *)
				MB_RegistriLetti[201] := ModBus.MB_Resp.Data[1];		(* Vedi tabella *)
				MB_RegistriLetti[202] := ModBus.MB_Resp.Data[2];		(* Vedi tabella *)
				MB_RegistriLetti[203] := ModBus.MB_Resp.Data[3];		(* Vedi tabella *)
				MB_RegistriLetti[204] := ModBus.MB_Resp.Data[4];		(* Vedi tabella *)
				MB_RegistriLetti[205] := ModBus.MB_Resp.Data[5];		(* Vedi tabella *)
				MB_RegistriLetti[206] := ModBus.MB_Resp.Data[6];		(* Vedi tabella *)
				MB_RegistriLetti[207] := ModBus.MB_Resp.Data[7];		(* Vedi tabella *)

				ModBus.MB_Query.Read_StartAddress := 209; (* richiedo lettura altri Parametri *)
				ModBus.MB_Query.Read_Quantity := 20;
				ModBus.MB_Start := TRUE;

				state := 55;
			END_IF
		END_IF

	55: (* Rispota Altri paramenti *)
		IF NOT ModBus.MB_Start  THEN

			IF ModBus.MB_MASTER.MB_Error<>0 THEN
				state := 300;
			ELSE
				MB_RegistriLetti[209] := ModBus.MB_Resp.Data[0];   	(* Vedi tabella *)
				MB_RegistriLetti[210] := ModBus.MB_Resp.Data[1];		(* Vedi tabella *)
				MB_RegistriLetti[211] := ModBus.MB_Resp.Data[2];		(* Vedi tabella *)
				MB_RegistriLetti[212] := ModBus.MB_Resp.Data[3];		(* Vedi tabella *)
				MB_RegistriLetti[213] := ModBus.MB_Resp.Data[4];		(* Vedi tabella *)
				MB_RegistriLetti[214] := ModBus.MB_Resp.Data[5];		(* Vedi tabella *)
				MB_RegistriLetti[215] := ModBus.MB_Resp.Data[6];		(* Vedi tabella *)
				MB_RegistriLetti[216] := ModBus.MB_Resp.Data[7];		(* Vedi tabella *)
				MB_RegistriLetti[217] := ModBus.MB_Resp.Data[8];		(* Vedi tabella *)
				MB_RegistriLetti[218] := ModBus.MB_Resp.Data[9];		(* Vedi tabella *)
				MB_RegistriLetti[219] := ModBus.MB_Resp.Data[10];		(* Vedi tabella *)
				MB_RegistriLetti[220] := ModBus.MB_Resp.Data[11];		(* Vedi tabella *)
				MB_RegistriLetti[221] := ModBus.MB_Resp.Data[12];		(* Vedi tabella *)
				MB_RegistriLetti[222] := ModBus.MB_Resp.Data[13];		(* Vedi tabella *)
				MB_RegistriLetti[223] := ModBus.MB_Resp.Data[14];		(* Vedi tabella *)
				MB_RegistriLetti[224] := ModBus.MB_Resp.Data[15];		(* Vedi tabella *)
				MB_RegistriLetti[225] := ModBus.MB_Resp.Data[16];		(* Vedi tabella *)
				MB_RegistriLetti[226] := ModBus.MB_Resp.Data[17];		(* Vedi tabella *)
				MB_RegistriLetti[227] := ModBus.MB_Resp.Data[18];		(* Vedi tabella *)
				MB_RegistriLetti[228] := ModBus.MB_Resp.Data[19];		(* Vedi tabella *)

				ModBus.MB_Query.Read_StartAddress := 229; (* richiedo lettura altri Parametri *)
				ModBus.MB_Query.Read_Quantity := 4;
				ModBus.MB_Start := TRUE;

				state := 60;
			END_IF
		END_IF

	60: (* Rispota Altri paramenti *)
		IF NOT ModBus.MB_Start  THEN

			IF ModBus.MB_MASTER.MB_Error<>0 THEN
				state := 300;
			ELSE
				MB_RegistriLetti[229] := ModBus.MB_Resp.Data[0];   	(* Vedi tabella *)
				MB_RegistriLetti[230] := ModBus.MB_Resp.Data[1];		(* Vedi tabella *)
				MB_RegistriLetti[231] := ModBus.MB_Resp.Data[2];		(* Vedi tabella *)
				MB_RegistriLetti[232] := ModBus.MB_Resp.Data[3];		(* Vedi tabella *)

				ModBus.MB_Query.Read_StartAddress := 235; (* richiedo lettura altri Parametri *)
				ModBus.MB_Query.Read_Quantity := 10;
				ModBus.MB_Start := TRUE;

				state := 65;
			END_IF
		END_IF


	65: (* Rispota Altri paramenti *)
		IF NOT ModBus.MB_Start  THEN

			IF ModBus.MB_MASTER.MB_Error<>0 THEN
				state := 300;
			ELSE
				MB_RegistriLetti[235] := ModBus.MB_Resp.Data[0];   	(* Vedi tabella *)
				MB_RegistriLetti[236] := ModBus.MB_Resp.Data[1];		(* Vedi tabella *)
				MB_RegistriLetti[237] := ModBus.MB_Resp.Data[2];		(* Vedi tabella *)
				MB_RegistriLetti[238] := ModBus.MB_Resp.Data[3];		(* Vedi tabella *)
				MB_RegistriLetti[239] := ModBus.MB_Resp.Data[4];		(* Vedi tabella *)
				MB_RegistriLetti[240] := ModBus.MB_Resp.Data[5];		(* Vedi tabella *)
				MB_RegistriLetti[241] := ModBus.MB_Resp.Data[6];		(* Vedi tabella *)
				MB_RegistriLetti[242] := ModBus.MB_Resp.Data[7];		(* Vedi tabella *)
				MB_RegistriLetti[243] := ModBus.MB_Resp.Data[8];		(* Vedi tabella *)
				MB_RegistriLetti[244] := ModBus.MB_Resp.Data[9];		(* Vedi tabella *)

				ModBus.MB_Query.Read_StartAddress := 268; (* richiedo lettura altri Parametri *)
				ModBus.MB_Query.Read_Quantity := 9;
				ModBus.MB_Start := TRUE;

				state := 70;
			END_IF
		END_IF

	70: (* Rispota Altri paramenti *)
		IF NOT ModBus.MB_Start  THEN

			IF ModBus.MB_MASTER.MB_Error<>0 THEN
				state := 300;
			ELSE
				MB_RegistriLetti[235] := ModBus.MB_Resp.Data[0];   	(* Vedi tabella *)
				MB_RegistriLetti[236] := ModBus.MB_Resp.Data[1];		(* Vedi tabella *)
				MB_RegistriLetti[237] := ModBus.MB_Resp.Data[2];		(* Vedi tabella *)
				MB_RegistriLetti[238] := ModBus.MB_Resp.Data[3];		(* Vedi tabella *)
				MB_RegistriLetti[239] := ModBus.MB_Resp.Data[4];		(* Vedi tabella *)
				MB_RegistriLetti[240] := ModBus.MB_Resp.Data[5];		(* Vedi tabella *)
				MB_RegistriLetti[241] := ModBus.MB_Resp.Data[6];		(* Vedi tabella *)
				MB_RegistriLetti[242] := ModBus.MB_Resp.Data[7];		(* Vedi tabella *)
				MB_RegistriLetti[243] := ModBus.MB_Resp.Data[8];		(* Vedi tabella *)
				MB_RegistriLetti[244] := ModBus.MB_Resp.Data[9];		(* Vedi tabella *)

				ModBus.MB_Query.Read_StartAddress := 268; (* richiedo lettura altri Parametri *)
				ModBus.MB_Query.Read_Quantity := 9;
				ModBus.MB_Start := TRUE;

				state := 75;
			END_IF
		END_IF


	75: (* Rispota Altri paramenti *)
		IF NOT ModBus.MB_Start  THEN

			IF ModBus.MB_MASTER.MB_Error<>0 THEN
				state := 300;
			ELSE
				MB_RegistriLetti[268] := ModBus.MB_Resp.Data[0];   	(* Vedi tabella *)
				MB_RegistriLetti[269] := ModBus.MB_Resp.Data[1];		(* Vedi tabella *)
				MB_RegistriLetti[270] := ModBus.MB_Resp.Data[2];		(* Vedi tabella *)
				MB_RegistriLetti[271] := ModBus.MB_Resp.Data[3];		(* Vedi tabella *)
				MB_RegistriLetti[272] := ModBus.MB_Resp.Data[4];		(* Vedi tabella *)
				MB_RegistriLetti[273] := ModBus.MB_Resp.Data[5];		(* Vedi tabella *)
				MB_RegistriLetti[274] := ModBus.MB_Resp.Data[6];		(* Vedi tabella *)
				MB_RegistriLetti[275] := ModBus.MB_Resp.Data[7];		(* Vedi tabella *)
				MB_RegistriLetti[276] := ModBus.MB_Resp.Data[8];		(* Vedi tabella *)

				ModBus.MB_Query.Read_StartAddress := 408; (* richiedo lettura altri Parametri *)
				ModBus.MB_Query.Read_Quantity := 6;
				ModBus.MB_Start := TRUE;

				state := 80;
			END_IF
		END_IF

	80: (* Rispota Altri paramenti *)
		IF NOT ModBus.MB_Start  THEN

			IF ModBus.MB_MASTER.MB_Error<>0 THEN
				state := 300;
			ELSE
				MB_RegistriLetti[408] := ModBus.MB_Resp.Data[0];   		(* Vedi tabella *)
				MB_RegistriLetti[409] := ModBus.MB_Resp.Data[1];		(* Vedi tabella *)
				MB_RegistriLetti[410] := ModBus.MB_Resp.Data[2];		(* Vedi tabella *)
				MB_RegistriLetti[411] := ModBus.MB_Resp.Data[3];		(* Vedi tabella *)
				MB_RegistriLetti[412] := ModBus.MB_Resp.Data[4];		(* Vedi tabella *)
				MB_RegistriLetti[413] := ModBus.MB_Resp.Data[5];		(* Vedi tabella *)

				ModBus.MB_Query.Read_StartAddress := 408; (* richiedo lettura altri Parametri *)
				ModBus.MB_Query.Read_Quantity := 6;
				ModBus.MB_Start := TRUE;

				state := 100;
			END_IF
		END_IF






	100: (* Rispota Altri paramenti COIL *)
		IF NOT ModBus.MB_Start  THEN

			IF ModBus.MB_MASTER.MB_Error<>0 THEN
				state := 300;
			ELSE
				Modbus.MB_Query.SlaveAddress := Address;
				Modbus.MB_Query.FunctionCode := 1;
				ModBus.MB_Query.Read_StartAddress := 0;	(* richiedo lettura altri Parametri *)
				ModBus.MB_Query.Read_Quantity := 60;
				ModBus.MB_Start := TRUE;

				state:=105;
			END_IF
		END_IF
	105: (* Rispota Altri paramenti *)

		IF NOT ModBus.MB_Start  THEN

			IF ModBus.MB_MASTER.MB_Error<>0 THEN
				state := 300;
			ELSE

				MB_BitStato[1]:=ModBus.MB_MASTER.ReceiveBuffer.Data[3].0; (*Vedi Tabella *)
				MB_BitStato[2]:=ModBus.MB_MASTER.ReceiveBuffer.Data[3].1; (*Vedi Tabella *)
				MB_BitStato[3]:=ModBus.MB_MASTER.ReceiveBuffer.Data[3].2; (*Vedi Tabella *)
				MB_BitStato[4]:=ModBus.MB_MASTER.ReceiveBuffer.Data[3].3; (*Vedi Tabella *)
				MB_BitStato[5]:=ModBus.MB_MASTER.ReceiveBuffer.Data[3].4; (*Vedi Tabella *)
				MB_BitStato[6]:=ModBus.MB_MASTER.ReceiveBuffer.Data[3].5; (*Vedi Tabella *)
				MB_BitStato[7]:=ModBus.MB_MASTER.ReceiveBuffer.Data[3].6; (*Vedi Tabella *)
				MB_BitStato[8]:=ModBus.MB_MASTER.ReceiveBuffer.Data[3].7; (*Vedi Tabella *)
				MB_BitStato[9]:=ModBus.MB_MASTER.ReceiveBuffer.Data[4].0; (*Vedi Tabella *)
				MB_BitStato[10]:=ModBus.MB_MASTER.ReceiveBuffer.Data[4].1; (*Vedi Tabella *)
				MB_BitStato[11]:=ModBus.MB_MASTER.ReceiveBuffer.Data[4].2; (*Vedi Tabella *)
				MB_BitStato[12]:=ModBus.MB_MASTER.ReceiveBuffer.Data[4].3; (*Vedi Tabella *)
				MB_BitStato[13]:=ModBus.MB_MASTER.ReceiveBuffer.Data[4].4; (*Vedi Tabella *)
				MB_BitStato[14]:=ModBus.MB_MASTER.ReceiveBuffer.Data[4].5; (*Vedi Tabella *)
				MB_BitStato[15]:=ModBus.MB_MASTER.ReceiveBuffer.Data[4].6; (*Vedi Tabella *)
				MB_BitStato[16]:=ModBus.MB_MASTER.ReceiveBuffer.Data[4].7; (*Vedi Tabella *)
				MB_BitStato[17]:=ModBus.MB_MASTER.ReceiveBuffer.Data[5].0; (*Vedi Tabella *)
				MB_BitStato[18]:=ModBus.MB_MASTER.ReceiveBuffer.Data[5].1; (*Vedi Tabella *)
				MB_BitStato[19]:=ModBus.MB_MASTER.ReceiveBuffer.Data[5].2; (*Vedi Tabella *)
				MB_BitStato[20]:=ModBus.MB_MASTER.ReceiveBuffer.Data[5].3; (*Vedi Tabella *)
				MB_BitStato[21]:=ModBus.MB_MASTER.ReceiveBuffer.Data[5].4; (*Vedi Tabella *)
				MB_BitStato[22]:=ModBus.MB_MASTER.ReceiveBuffer.Data[5].5; (*Vedi Tabella *)
				MB_BitStato[23]:=ModBus.MB_MASTER.ReceiveBuffer.Data[5].6; (*Vedi Tabella *)
				MB_BitStato[24]:=ModBus.MB_MASTER.ReceiveBuffer.Data[5].7; (*Vedi Tabella *)
				MB_BitStato[25]:=ModBus.MB_MASTER.ReceiveBuffer.Data[6].0; (*Vedi Tabella *)
				MB_BitStato[26]:=ModBus.MB_MASTER.ReceiveBuffer.Data[6].1; (*Vedi Tabella *)
				MB_BitStato[27]:=ModBus.MB_MASTER.ReceiveBuffer.Data[6].2; (*Vedi Tabella *)
				MB_BitStato[28]:=ModBus.MB_MASTER.ReceiveBuffer.Data[6].3; (*Vedi Tabella *)
				MB_BitStato[29]:=ModBus.MB_MASTER.ReceiveBuffer.Data[6].4; (*Vedi Tabella *)
				MB_BitStato[30]:=ModBus.MB_MASTER.ReceiveBuffer.Data[6].5; (*Vedi Tabella *)
				MB_BitStato[31]:=ModBus.MB_MASTER.ReceiveBuffer.Data[6].6; (*Vedi Tabella *)
				MB_BitStato[32]:=ModBus.MB_MASTER.ReceiveBuffer.Data[6].7; (*Vedi Tabella *)
				MB_BitStato[33]:=ModBus.MB_MASTER.ReceiveBuffer.Data[7].0; (*Vedi Tabella *)
				MB_BitStato[34]:=ModBus.MB_MASTER.ReceiveBuffer.Data[7].1; (*Vedi Tabella *)
				MB_BitStato[35]:=ModBus.MB_MASTER.ReceiveBuffer.Data[7].2; (*Vedi Tabella *)
				MB_BitStato[36]:=ModBus.MB_MASTER.ReceiveBuffer.Data[7].3; (*Vedi Tabella *)
				MB_BitStato[37]:=ModBus.MB_MASTER.ReceiveBuffer.Data[7].4; (*Vedi Tabella *)
				MB_BitStato[38]:=ModBus.MB_MASTER.ReceiveBuffer.Data[7].5; (*Vedi Tabella *)
				MB_BitStato[39]:=ModBus.MB_MASTER.ReceiveBuffer.Data[7].6; (*Vedi Tabella *)
				MB_BitStato[40]:=ModBus.MB_MASTER.ReceiveBuffer.Data[7].7; (*Vedi Tabella *)
				MB_BitStato[41]:=ModBus.MB_MASTER.ReceiveBuffer.Data[8].0; (*Vedi Tabella *)
				MB_BitStato[42]:=ModBus.MB_MASTER.ReceiveBuffer.Data[8].1; (*Vedi Tabella *)
				MB_BitStato[43]:=ModBus.MB_MASTER.ReceiveBuffer.Data[8].2; (*Vedi Tabella *)
				MB_BitStato[44]:=ModBus.MB_MASTER.ReceiveBuffer.Data[8].3; (*Vedi Tabella *)
				MB_BitStato[45]:=ModBus.MB_MASTER.ReceiveBuffer.Data[8].4; (*Vedi Tabella *)
				MB_BitStato[46]:=ModBus.MB_MASTER.ReceiveBuffer.Data[8].5; (*Vedi Tabella *)
				MB_BitStato[47]:=ModBus.MB_MASTER.ReceiveBuffer.Data[8].6; (*Vedi Tabella *)
				MB_BitStato[48]:=ModBus.MB_MASTER.ReceiveBuffer.Data[8].7; (*Vedi Tabella *)
				MB_BitStato[49]:=ModBus.MB_MASTER.ReceiveBuffer.Data[9].0; (*Vedi Tabella *)
				MB_BitStato[50]:=ModBus.MB_MASTER.ReceiveBuffer.Data[9].1; (*Vedi Tabella *)
				MB_BitStato[51]:=ModBus.MB_MASTER.ReceiveBuffer.Data[9].2; (*Vedi Tabella *)
				MB_BitStato[52]:=ModBus.MB_MASTER.ReceiveBuffer.Data[9].3; (*Vedi Tabella *)
				MB_BitStato[53]:=ModBus.MB_MASTER.ReceiveBuffer.Data[9].4; (*Vedi Tabella *)
				MB_BitStato[54]:=ModBus.MB_MASTER.ReceiveBuffer.Data[9].5; (*Vedi Tabella *)
				MB_BitStato[55]:=ModBus.MB_MASTER.ReceiveBuffer.Data[9].6; (*Vedi Tabella *)
				MB_BitStato[56]:=ModBus.MB_MASTER.ReceiveBuffer.Data[9].7; (*Vedi Tabella *)
				MB_BitStato[57]:=ModBus.MB_MASTER.ReceiveBuffer.Data[10].0; (*Vedi Tabella *)
				MB_BitStato[58]:=ModBus.MB_MASTER.ReceiveBuffer.Data[10].1; (*Vedi Tabella *)
				MB_BitStato[59]:=ModBus.MB_MASTER.ReceiveBuffer.Data[10].2; (*Vedi Tabella *)
				MB_BitStato[60]:=ModBus.MB_MASTER.ReceiveBuffer.Data[10].3; (*Vedi Tabella *)
				MB_BitStato[61]:=ModBus.MB_MASTER.ReceiveBuffer.Data[10].4; (*Vedi Tabella *)
				MB_BitStato[62]:=ModBus.MB_MASTER.ReceiveBuffer.Data[10].5; (*Vedi Tabella *)
				MB_BitStato[63]:=ModBus.MB_MASTER.ReceiveBuffer.Data[10].6; (*Vedi Tabella *)
				MB_BitStato[64]:=ModBus.MB_MASTER.ReceiveBuffer.Data[10].7; (*Vedi Tabella *)


				state:=110;

			END_IF
		END_IF


	110: (* Rispota Altri paramenti *)
		IF NOT ModBus.MB_Start  THEN

			IF ModBus.MB_MASTER.MB_Error<>0 THEN
				state := 300;
			ELSE
				Modbus.MB_Query.SlaveAddress := Address;
				Modbus.MB_Query.FunctionCode := 1;
				ModBus.MB_Query.Read_StartAddress := 100;
				ModBus.MB_Query.Read_Quantity := 100;
				ModBus.MB_Start := TRUE;

				state:=115;
			END_IF
		END_IF
	115: (* Rispota Altri paramenti *)

		IF NOT ModBus.MB_Start  THEN

			IF ModBus.MB_MASTER.MB_Error<>0 THEN
				state := 300;
			ELSE

				MB_BitStato[100]:=ModBus.MB_MASTER.ReceiveBuffer.Data[3].0; (*Vedi Tabella *)
				MB_BitStato[101]:=ModBus.MB_MASTER.ReceiveBuffer.Data[3].1; (*Vedi Tabella *)
				MB_BitStato[102]:=ModBus.MB_MASTER.ReceiveBuffer.Data[3].2; (*Vedi Tabella *)
				MB_BitStato[103]:=ModBus.MB_MASTER.ReceiveBuffer.Data[3].3; (*Vedi Tabella *)
				MB_BitStato[104]:=ModBus.MB_MASTER.ReceiveBuffer.Data[3].4; (*Vedi Tabella *)
				MB_BitStato[105]:=ModBus.MB_MASTER.ReceiveBuffer.Data[3].5; (*Vedi Tabella *)
				MB_BitStato[106]:=ModBus.MB_MASTER.ReceiveBuffer.Data[3].6; (*Vedi Tabella *)
				MB_BitStato[107]:=ModBus.MB_MASTER.ReceiveBuffer.Data[3].7; (*Vedi Tabella *)
				MB_BitStato[108]:=ModBus.MB_MASTER.ReceiveBuffer.Data[4].0; (*Vedi Tabella *)
				MB_BitStato[109]:=ModBus.MB_MASTER.ReceiveBuffer.Data[4].1; (*Vedi Tabella *)
				MB_BitStato[110]:=ModBus.MB_MASTER.ReceiveBuffer.Data[4].2; (*Vedi Tabella *)
				MB_BitStato[111]:=ModBus.MB_MASTER.ReceiveBuffer.Data[4].3; (*Vedi Tabella *)
				MB_BitStato[112]:=ModBus.MB_MASTER.ReceiveBuffer.Data[4].4; (*Vedi Tabella *)
				MB_BitStato[113]:=ModBus.MB_MASTER.ReceiveBuffer.Data[4].5; (*Vedi Tabella *)
				MB_BitStato[114]:=ModBus.MB_MASTER.ReceiveBuffer.Data[4].6; (*Vedi Tabella *)
				MB_BitStato[115]:=ModBus.MB_MASTER.ReceiveBuffer.Data[4].7; (*Vedi Tabella *)
				MB_BitStato[116]:=ModBus.MB_MASTER.ReceiveBuffer.Data[5].0; (*Vedi Tabella *)
				MB_BitStato[117]:=ModBus.MB_MASTER.ReceiveBuffer.Data[5].1; (*Vedi Tabella *)
				MB_BitStato[118]:=ModBus.MB_MASTER.ReceiveBuffer.Data[5].2; (*Vedi Tabella *)
				MB_BitStato[119]:=ModBus.MB_MASTER.ReceiveBuffer.Data[5].3; (*Vedi Tabella *)
				MB_BitStato[120]:=ModBus.MB_MASTER.ReceiveBuffer.Data[5].4; (*Vedi Tabella *)
				MB_BitStato[121]:=ModBus.MB_MASTER.ReceiveBuffer.Data[5].5; (*Vedi Tabella *)
				MB_BitStato[122]:=ModBus.MB_MASTER.ReceiveBuffer.Data[5].6; (*Vedi Tabella *)
				MB_BitStato[123]:=ModBus.MB_MASTER.ReceiveBuffer.Data[5].7; (*Vedi Tabella *)
				MB_BitStato[124]:=ModBus.MB_MASTER.ReceiveBuffer.Data[6].0; (*Vedi Tabella *)
				MB_BitStato[125]:=ModBus.MB_MASTER.ReceiveBuffer.Data[6].1; (*Vedi Tabella *)
				MB_BitStato[126]:=ModBus.MB_MASTER.ReceiveBuffer.Data[6].2; (*Vedi Tabella *)
				MB_BitStato[127]:=ModBus.MB_MASTER.ReceiveBuffer.Data[6].3; (*Vedi Tabella *)
				MB_BitStato[128]:=ModBus.MB_MASTER.ReceiveBuffer.Data[6].4; (*Vedi Tabella *)
				MB_BitStato[129]:=ModBus.MB_MASTER.ReceiveBuffer.Data[6].5; (*Vedi Tabella *)
				MB_BitStato[130]:=ModBus.MB_MASTER.ReceiveBuffer.Data[6].6; (*Vedi Tabella *)
				MB_BitStato[131]:=ModBus.MB_MASTER.ReceiveBuffer.Data[6].7; (*Vedi Tabella *)
				MB_BitStato[132]:=ModBus.MB_MASTER.ReceiveBuffer.Data[7].0; (*Vedi Tabella *)
				MB_BitStato[133]:=ModBus.MB_MASTER.ReceiveBuffer.Data[7].1; (*Vedi Tabella *)
				MB_BitStato[134]:=ModBus.MB_MASTER.ReceiveBuffer.Data[7].2; (*Vedi Tabella *)
				MB_BitStato[135]:=ModBus.MB_MASTER.ReceiveBuffer.Data[7].3; (*Vedi Tabella *)
				MB_BitStato[136]:=ModBus.MB_MASTER.ReceiveBuffer.Data[7].4; (*Vedi Tabella *)
				MB_BitStato[137]:=ModBus.MB_MASTER.ReceiveBuffer.Data[7].5; (*Vedi Tabella *)
				MB_BitStato[138]:=ModBus.MB_MASTER.ReceiveBuffer.Data[7].6; (*Vedi Tabella *)
				MB_BitStato[139]:=ModBus.MB_MASTER.ReceiveBuffer.Data[7].7; (*Vedi Tabella *)
				MB_BitStato[140]:=ModBus.MB_MASTER.ReceiveBuffer.Data[8].0; (*Vedi Tabella *)
				MB_BitStato[141]:=ModBus.MB_MASTER.ReceiveBuffer.Data[8].1; (*Vedi Tabella *)
				MB_BitStato[142]:=ModBus.MB_MASTER.ReceiveBuffer.Data[8].2; (*Vedi Tabella *)
				MB_BitStato[143]:=ModBus.MB_MASTER.ReceiveBuffer.Data[8].3; (*Vedi Tabella *)
				MB_BitStato[144]:=ModBus.MB_MASTER.ReceiveBuffer.Data[8].4; (*Vedi Tabella *)
				MB_BitStato[145]:=ModBus.MB_MASTER.ReceiveBuffer.Data[8].5; (*Vedi Tabella *)
				MB_BitStato[146]:=ModBus.MB_MASTER.ReceiveBuffer.Data[8].6; (*Vedi Tabella *)
				MB_BitStato[147]:=ModBus.MB_MASTER.ReceiveBuffer.Data[8].7; (*Vedi Tabella *)
				MB_BitStato[148]:=ModBus.MB_MASTER.ReceiveBuffer.Data[9].0; (*Vedi Tabella *)
				MB_BitStato[149]:=ModBus.MB_MASTER.ReceiveBuffer.Data[9].1; (*Vedi Tabella *)
				MB_BitStato[150]:=ModBus.MB_MASTER.ReceiveBuffer.Data[9].2; (*Vedi Tabella *)
				MB_BitStato[151]:=ModBus.MB_MASTER.ReceiveBuffer.Data[9].3; (*Vedi Tabella *)
				MB_BitStato[152]:=ModBus.MB_MASTER.ReceiveBuffer.Data[9].4; (*Vedi Tabella *)
				MB_BitStato[153]:=ModBus.MB_MASTER.ReceiveBuffer.Data[9].5; (*Vedi Tabella *)
				MB_BitStato[154]:=ModBus.MB_MASTER.ReceiveBuffer.Data[9].6; (*Vedi Tabella *)
				MB_BitStato[155]:=ModBus.MB_MASTER.ReceiveBuffer.Data[9].7; (*Vedi Tabella *)
				MB_BitStato[156]:=ModBus.MB_MASTER.ReceiveBuffer.Data[10].0; (*Vedi Tabella *)
				MB_BitStato[157]:=ModBus.MB_MASTER.ReceiveBuffer.Data[10].1; (*Vedi Tabella *)
				MB_BitStato[158]:=ModBus.MB_MASTER.ReceiveBuffer.Data[10].2; (*Vedi Tabella *)
				MB_BitStato[159]:=ModBus.MB_MASTER.ReceiveBuffer.Data[10].3; (*Vedi Tabella *)
				MB_BitStato[160]:=ModBus.MB_MASTER.ReceiveBuffer.Data[10].4; (*Vedi Tabella *)
				MB_BitStato[161]:=ModBus.MB_MASTER.ReceiveBuffer.Data[10].5; (*Vedi Tabella *)
				MB_BitStato[162]:=ModBus.MB_MASTER.ReceiveBuffer.Data[10].6; (*Vedi Tabella *)
				MB_BitStato[163]:=ModBus.MB_MASTER.ReceiveBuffer.Data[10].7; (*Vedi Tabella *)
				MB_BitStato[164]:=ModBus.MB_MASTER.ReceiveBuffer.Data[11].0; (*Vedi Tabella *)
				MB_BitStato[165]:=ModBus.MB_MASTER.ReceiveBuffer.Data[11].1; (*Vedi Tabella *)
				MB_BitStato[166]:=ModBus.MB_MASTER.ReceiveBuffer.Data[11].2; (*Vedi Tabella *)
				MB_BitStato[167]:=ModBus.MB_MASTER.ReceiveBuffer.Data[11].3; (*Vedi Tabella *)
				MB_BitStato[168]:=ModBus.MB_MASTER.ReceiveBuffer.Data[11].4; (*Vedi Tabella *)
				MB_BitStato[169]:=ModBus.MB_MASTER.ReceiveBuffer.Data[11].5; (*Vedi Tabella *)
				MB_BitStato[170]:=ModBus.MB_MASTER.ReceiveBuffer.Data[11].6; (*Vedi Tabella *)
				MB_BitStato[171]:=ModBus.MB_MASTER.ReceiveBuffer.Data[11].7; (*Vedi Tabella *)
				MB_BitStato[172]:=ModBus.MB_MASTER.ReceiveBuffer.Data[12].0; (*Vedi Tabella *)
				MB_BitStato[173]:=ModBus.MB_MASTER.ReceiveBuffer.Data[12].1; (*Vedi Tabella *)
				MB_BitStato[174]:=ModBus.MB_MASTER.ReceiveBuffer.Data[12].2; (*Vedi Tabella *)
				MB_BitStato[175]:=ModBus.MB_MASTER.ReceiveBuffer.Data[12].3; (*Vedi Tabella *)
				MB_BitStato[176]:=ModBus.MB_MASTER.ReceiveBuffer.Data[12].4; (*Vedi Tabella *)
				MB_BitStato[177]:=ModBus.MB_MASTER.ReceiveBuffer.Data[12].5; (*Vedi Tabella *)
				MB_BitStato[178]:=ModBus.MB_MASTER.ReceiveBuffer.Data[12].6; (*Vedi Tabella *)
				MB_BitStato[179]:=ModBus.MB_MASTER.ReceiveBuffer.Data[12].7; (*Vedi Tabella *)
				MB_BitStato[180]:=ModBus.MB_MASTER.ReceiveBuffer.Data[13].0; (*Vedi Tabella *)
				MB_BitStato[181]:=ModBus.MB_MASTER.ReceiveBuffer.Data[13].1; (*Vedi Tabella *)
				MB_BitStato[182]:=ModBus.MB_MASTER.ReceiveBuffer.Data[13].2; (*Vedi Tabella *)
				MB_BitStato[183]:=ModBus.MB_MASTER.ReceiveBuffer.Data[13].3; (*Vedi Tabella *)
				MB_BitStato[184]:=ModBus.MB_MASTER.ReceiveBuffer.Data[13].4; (*Vedi Tabella *)
				MB_BitStato[185]:=ModBus.MB_MASTER.ReceiveBuffer.Data[13].5; (*Vedi Tabella *)
				MB_BitStato[186]:=ModBus.MB_MASTER.ReceiveBuffer.Data[13].6; (*Vedi Tabella *)
				MB_BitStato[187]:=ModBus.MB_MASTER.ReceiveBuffer.Data[13].7; (*Vedi Tabella *)
				MB_BitStato[188]:=ModBus.MB_MASTER.ReceiveBuffer.Data[13].0; (*Vedi Tabella *)
				MB_BitStato[189]:=ModBus.MB_MASTER.ReceiveBuffer.Data[13].1; (*Vedi Tabella *)
				MB_BitStato[190]:=ModBus.MB_MASTER.ReceiveBuffer.Data[13].2; (*Vedi Tabella *)
				MB_BitStato[191]:=ModBus.MB_MASTER.ReceiveBuffer.Data[13].3; (*Vedi Tabella *)
				MB_BitStato[192]:=ModBus.MB_MASTER.ReceiveBuffer.Data[13].4; (*Vedi Tabella *)
				MB_BitStato[193]:=ModBus.MB_MASTER.ReceiveBuffer.Data[13].5; (*Vedi Tabella *)
				MB_BitStato[194]:=ModBus.MB_MASTER.ReceiveBuffer.Data[13].6; (*Vedi Tabella *)
				MB_BitStato[195]:=ModBus.MB_MASTER.ReceiveBuffer.Data[13].7; (*Vedi Tabella *)
				MB_BitStato[196]:=ModBus.MB_MASTER.ReceiveBuffer.Data[14].0; (*Vedi Tabella *)
				MB_BitStato[197]:=ModBus.MB_MASTER.ReceiveBuffer.Data[14].1; (*Vedi Tabella *)
				MB_BitStato[198]:=ModBus.MB_MASTER.ReceiveBuffer.Data[14].2; (*Vedi Tabella *)
				MB_BitStato[199]:=ModBus.MB_MASTER.ReceiveBuffer.Data[14].3; (*Vedi Tabella *)


				state:=200;

			END_IF
		END_IF


	200:
		IF NOT ModBus.MB_Start  THEN

			IF ModBus.MB_MASTER.MB_Error<>0 THEN
				state := 300;
			ELSE
				IF ScriviDato THEN
					state := 205;
				ELSE
					state := 295;
				END_IF
			END_IF
		END_IF


	 205:	(* Scrivo la Variabile all'indirizzo specificato  *)

		Modbus.MB_Query.SlaveAddress := Address;
		Modbus.MB_Query.FunctionCode := 6;
		ModBus.MB_Query.Write_StartAddress := IndirizzoDaScrivere;
		ModBus.MB_Query.Write_Quantity :=1;
		ModBus.MB_Query.Write_Data[0] := DatoDaScrivere;
		ModBus.MB_Start := TRUE;

		state := 295;



		295:
		IF NOT ModBus.MB_Start THEN
			IF ModBus.MB_MASTER.MB_Error<>0 THEN (*OR ModBus.MB_MASTER.MB_Error<>0 THEN*)
				state := 300;
			ELSE
				IF fModbusAlr THEN fModbusAlr := FALSE; END_IF
				NodoDaInterrogareChiller:=Address+1;
				InibiscoModbusChiller:=FALSE;
				retryErr := 0;
				retry := 0;
				state := 0;
					IF fModbusAlr=FALSE AND ErroreComuModBus=TRUE THEN
						LogEv(EL_Log,EO_CHI,ID,62,'ComunicazioneModBus_OK');
						ErroreComuModBus := FALSE;
				(*	WarningCtr := SEL(WarningCtr=0, WarningCtr-1, 0); *)
					END_IF


			END_IF
		END_IF



	(**** CHECK MODBUS ERROR ****)
	300: 	(* Release MODBUS *)
			InibiscoModbusChiller:=FALSE;
			(* Retries *)
			retry:=retry+1;
			IF retry>3 THEN
				retry:=0;

				(* Verify if slave is dead *)
				IF retryErr < retryErrMaX THEN
					retryErr := retryErr + 1;
				ELSE
					fModbusAlr := TRUE;
					(* Verify ModBus error	*)

					IF fModbusAlr AND ErroreComuModBus=FALSE THEN
						LogEv(EL_Alarm,EO_CHI,ID,61,CONCAT('ErroreModbus_',INT_TO_STRING(ModBus.MB_MASTER.MB_Error)));
						ErroreComuModBus := TRUE;
					END_IF
				END_IF

				END_IF
			Refresh_Now := FALSE;
			NodoDaInterrogareChiller:=Address+1;
			state:=0;
END_CASE




(* Controllo Time Out Ciclo ModBus *)

TimeOutModBus(In:=state<>0,PT:=t#30s);
IF TimeOutModBus.Q THEN
	State:=0;
	Refresh_Now:=TRUE;  (* Rilancio la lettura del nodo *)
	IF MODBUS.MB_Lock=TRUE THEN MODBUS.MB_Lock:=FALSE;END_IF
	IF InibiscoModbusChiller=TRUE THEN InibiscoModbusChiller:=FALSE;END_IF
END_IF
END_ACTION

(* POU Utils Functions/TONOF, ST *)
FUNCTION_BLOCK TONOF
VAR_INPUT
	IN		: BOOL;
	PT_ON	: TIME; (* time to pass, before OUT is set *)
	PT_OF	: TIME; (* time to pass, before OUT is reset *)
END_VAR
VAR_OUTPUT
	OUT		: BOOL;
END_VAR
VAR
	timer	: TON;
END_VAR
IF IN<>OUT THEN
	timer(IN:=TRUE,PT:=SEL(IN,PT_OF,PT_ON));
	IF timer.Q THEN OUT:=IN; END_IF
ELSE
	timer(IN:=FALSE);
END_IF
END_FUNCTION_BLOCK

(* POU Plant_Objects/obj_MODBUS_TRENDCOIN_01, ST *)
FUNCTION_BLOCK obj_MODBUS_TRENDCOIN_01
VAR CONSTANT

	TimeOutModBus: TON;


END_VAR
VAR_INPUT
	ID			:	BYTE;
	Address		:	BYTE;
	(* Modbus *)
	Refresh_Now	:	BOOL;			(* Richiesta di lettura stato macchina Immediata  *)
	retryErrMax	:	BYTE := 2;

(*	IndirizzoDaScrivere: WORD;
	DatoDaScrivere: INT;
	ScriviDato: BOOL; *)

END_VAR
VAR_IN_OUT
	ModBus		:obj_MODBUS;

END_VAR
VAR_OUTPUT
	Status_Log	:	WORD;
	Status_Vis	:	DWORD;
END_VAR
VAR

	state		:	INT;
	retry		:	BYTE;
	retryErr	:	BYTE;
	ReadTmr		:	TON := (PT:=T#5s);
	fModbusAlr:BOOL;

(*	retry_write	:	BYTE;
	fWriteStatus:	BOOL;
	fWriteMode	:	BOOL;
	fWriteReset	:	BOOL; *)

	x: INT;

	VerificaFuctionCode: INT;
	VerificaNodoLetto: INT;
	ErroreComuModBus: BOOL;
	IndiceErrore: BYTE;

	MB_BitStato: ARRAY [0..450] OF BOOL;
	MB_RegistriLetti: ARRAY [0..450] OF INT;

	MB_RegistriHoldingLetti: ARRAY [0..170] OF INT;
	MB_BitStatoCoil: ARRAY [0..100] OF BOOL;



	AddressRead: BYTE;
	index: BYTE;
	indexErr: BYTE;


	MB_V_L1_N: DWORD;
	MB_V_L2_N: DWORD;
	MB_V_L3_N: DWORD;
	MB_V_L1_L2: DWORD;
	MB_V_L1_L3: DWORD;
	MB_V_IL1: DWORD;
	MB_V_IL2: DWORD;
	MB_V_IL3: DWORD;
	MB_V_F: DWORD;
	MB_V_P: DWORD;
	MB_V_Q: DWORD;
	MB_V_P_F: DWORD;



	Read_StartAddress: INT;
	Read_Quantity: BYTE;
	IndiceMBLettura: INT;
	IndiceMBLetto: INT;
	test_Address: INT;
	Test_ScriviCoil: BOOL;
	test_Write: WORD;
	ScriviMB: BOOL;
END_VAR
(* Call ModBus state machine *)
Stm();

(* Check alarm	*)




(* Seganalzione stato Frigorifero  *)
IF ErroreComuModBus THEN
		Status_Log:=2; Status_Vis:=16#2020F0;
(*	ELSIF Warning OR Warning2 THEN
		Status_Log:=1; Status_Vis:=16#20F0F0; *)
    ELSE
		Status_Log:=0;
		Status_Vis:=16#006000;
END_IF
END_FUNCTION_BLOCK
ACTION AddLogData:
Logger.s1:=INSERT('&UTA=',BYTE_TO_STRING(ID),4);
IF ID<10 THEN Logger.s1:=INSERT(Logger.s1,'0',4); END_IF
(*

	Logger.s1:=CONCAT(Logger.s1,DWORD_TO_STRING(MB_V_L1_N));
	Logger.s1:=CONCAT(Logger.s1,';');
	Logger.s1:=CONCAT(Logger.s1,DWORD_TO_STRING(MB_V_L2_N));
	Logger.s1:=CONCAT(Logger.s1,';');
	Logger.s1:=CONCAT(Logger.s1,DWORD_TO_STRING(MB_V_L3_N));
	Logger.s1:=CONCAT(Logger.s1,';');
	Logger.s1:=CONCAT(Logger.s1,DWORD_TO_STRING(MB_V_L1_L2));
	Logger.s1:=CONCAT(Logger.s1,';');
	Logger.s1:=CONCAT(Logger.s1,DWORD_TO_STRING(MB_V_L1_L3));
	Logger.s1:=CONCAT(Logger.s1,';');
	Logger.s1:=CONCAT(Logger.s1,DWORD_TO_STRING(MB_V_IL1));
	Logger.s1:=CONCAT(Logger.s1,';');
	Logger.s1:=CONCAT(Logger.s1,DWORD_TO_STRING(MB_V_IL2));
	Logger.s1:=CONCAT(Logger.s1,';');
	Logger.s1:=CONCAT(Logger.s1,DWORD_TO_STRING(MB_V_IL3));
	Logger.s1:=CONCAT(Logger.s1,';');
	Logger.s1:=CONCAT(Logger.s1,DWORD_TO_STRING(MB_V_F));
	Logger.s1:=CONCAT(Logger.s1,';');
	Logger.s1:=CONCAT(Logger.s1,DWORD_TO_STRING(MB_V_P));
	Logger.s1:=CONCAT(Logger.s1,';');
	Logger.s1:=CONCAT(Logger.s1,DWORD_TO_STRING(MB_V_Q));
	Logger.s1:=CONCAT(Logger.s1,';');
	Logger.s1:=CONCAT(Logger.s1,DWORD_TO_STRING(MB_V_P_F));
*)


ADDSTRING(ADR(Logger.TData), ADR(Logger.s1), Logger.TLen);
END_ACTION
ACTION Stm:
CASE state OF
	0:	(* Refresh time manager *)
		ReadTmr(IN:=NOT ReadTmr.Q);
		(*A tempo interrogo il nodo sempre che non ci sia qualcuno che lo sta interrogando in quel momento *)

		IF (ReadTmr.Q AND NodoDaInterrogareMB1=Address )OR Refresh_Now AND NOT InibiscoModbusMB1 THEN
			state := 10;
			ReadTmr.PT := T#10s;  (* moreno *)
			Refresh_Now := FALSE;
			InibiscoModbusMB1 := TRUE;
		END_IF

	(**** Leggo le Analogiche a Disposzione  ****)

	10:	(* richiedo lettura di tutti gli Input Register   *)

		Modbus.MB_Query.SlaveAddress := Address;
		Modbus.MB_Query.FunctionCode := 4;
		Read_StartAddress := 0 ;			(* richiedo lettura altri Parametri *)
		Read_Quantity := 20;
		ModBus.MB_Start := TRUE;
		state := 20;


	20:
		ModBus.MB_Query.Read_StartAddress := 0 ;			(* richiedo lettura altri Parametri *)
		ModBus.MB_Query.Read_Quantity := 20;
		ModBus.MB_Start := TRUE;
		Read_StartAddress := 0 ;
		state := 30;



	30:	(* Risposta all'interrogazione *)
		IF NOT ModBus.MB_Start   THEN
			VerificaFuctionCode:=ModBus.MB_Resp.FunctionCode;
			VerificaNodoLetto:=ModBus.MB_Resp.SlaveAddress;

			IF ModBus.MB_MASTER.MB_Error<>0 THEN
				state := 300;
			ELSE

				FOR x:= 0 TO ModBus.MB_Query.Read_Quantity DO
					MB_RegistriLetti[Read_StartAddress+x ] := ModBus.MB_Resp.Data[x];   	(* Vedi tabella *)
				END_FOR

			ModBus.MB_Query.Read_StartAddress := 20 ;			(* richiedo lettura altri Parametri *)
			ModBus.MB_Query.Read_Quantity := 20;
			ModBus.MB_Start := TRUE;
			Read_StartAddress := 20 ;
			state := 31;
			END_IF
		END_IF


	31:	(* Risposta all'interrogazione *)
		IF NOT ModBus.MB_Start   THEN
			VerificaFuctionCode:=ModBus.MB_Resp.FunctionCode;
			VerificaNodoLetto:=ModBus.MB_Resp.SlaveAddress;

			IF ModBus.MB_MASTER.MB_Error<>0 THEN
				state := 300;
			ELSE

				FOR x:= 0 TO ModBus.MB_Query.Read_Quantity DO
					MB_RegistriLetti[Read_StartAddress+x ] := ModBus.MB_Resp.Data[x];   	(* Vedi tabella *)
				END_FOR

			ModBus.MB_Query.Read_StartAddress := 40 ;			(* richiedo lettura altri Parametri *)
			ModBus.MB_Query.Read_Quantity := 20;
			ModBus.MB_Start := TRUE;
			Read_StartAddress := 40 ;
			state := 32;
			END_IF
		END_IF



	32:	(* Risposta all'interrogazione *)
		IF NOT ModBus.MB_Start   THEN
			VerificaFuctionCode:=ModBus.MB_Resp.FunctionCode;
			VerificaNodoLetto:=ModBus.MB_Resp.SlaveAddress;

			IF ModBus.MB_MASTER.MB_Error<>0 THEN
				state := 300;
			ELSE

				FOR x:= 0 TO ModBus.MB_Query.Read_Quantity DO
					MB_RegistriLetti[Read_StartAddress+x ] := ModBus.MB_Resp.Data[x];   	(* Vedi tabella *)
				END_FOR

			ModBus.MB_Query.Read_StartAddress := 60 ;			(* richiedo lettura altri Parametri *)
			ModBus.MB_Query.Read_Quantity := 20;
			ModBus.MB_Start := TRUE;
			Read_StartAddress := 60 ;
			state := 33;
			END_IF
		END_IF

	33:	(* Risposta all'interrogazione *)
		IF NOT ModBus.MB_Start   THEN
			VerificaFuctionCode:=ModBus.MB_Resp.FunctionCode;
			VerificaNodoLetto:=ModBus.MB_Resp.SlaveAddress;

			IF ModBus.MB_MASTER.MB_Error<>0 THEN
				state := 300;
			ELSE

				FOR x:= 0 TO ModBus.MB_Query.Read_Quantity DO
					MB_RegistriLetti[Read_StartAddress+x ] := ModBus.MB_Resp.Data[x];   	(* Vedi tabella *)
				END_FOR

			ModBus.MB_Query.Read_StartAddress := 80 ;			(* richiedo lettura altri Parametri *)
			ModBus.MB_Query.Read_Quantity := 20;
			ModBus.MB_Start := TRUE;
			Read_StartAddress := 80 ;
			state := 34;
			END_IF
		END_IF


	34:	(* Risposta all'interrogazione *)
		IF NOT ModBus.MB_Start   THEN
			VerificaFuctionCode:=ModBus.MB_Resp.FunctionCode;
			VerificaNodoLetto:=ModBus.MB_Resp.SlaveAddress;

			IF ModBus.MB_MASTER.MB_Error<>0 THEN
				state := 300;
			ELSE

				FOR x:= 0 TO ModBus.MB_Query.Read_Quantity DO
					MB_RegistriLetti[Read_StartAddress+x ] := ModBus.MB_Resp.Data[x];   	(* Vedi tabella *)
				END_FOR

			ModBus.MB_Query.Read_StartAddress := 100 ;			(* richiedo lettura altri Parametri *)
			ModBus.MB_Query.Read_Quantity := 20;
			ModBus.MB_Start := TRUE;
			Read_StartAddress := 100 ;
			state := 35;
			END_IF
		END_IF


	35:	(* Risposta all'interrogazione *)
		IF NOT ModBus.MB_Start   THEN
			VerificaFuctionCode:=ModBus.MB_Resp.FunctionCode;
			VerificaNodoLetto:=ModBus.MB_Resp.SlaveAddress;

			IF ModBus.MB_MASTER.MB_Error<>0 THEN
				state := 300;
			ELSE

				FOR x:= 0 TO ModBus.MB_Query.Read_Quantity DO
					MB_RegistriLetti[Read_StartAddress+x ] := ModBus.MB_Resp.Data[x];   	(* Vedi tabella *)
				END_FOR

			ModBus.MB_Query.Read_StartAddress := 120 ;			(* richiedo lettura altri Parametri *)
			ModBus.MB_Query.Read_Quantity := 20;
			ModBus.MB_Start := TRUE;
			Read_StartAddress := 120 ;
			state := 36;
			END_IF
		END_IF

	36:	(* Risposta all'interrogazione *)
		IF NOT ModBus.MB_Start   THEN
			VerificaFuctionCode:=ModBus.MB_Resp.FunctionCode;
			VerificaNodoLetto:=ModBus.MB_Resp.SlaveAddress;

			IF ModBus.MB_MASTER.MB_Error<>0 THEN
				state := 300;
			ELSE

				FOR x:= 0 TO ModBus.MB_Query.Read_Quantity DO
					MB_RegistriLetti[Read_StartAddress+x ] := ModBus.MB_Resp.Data[x];   	(* Vedi tabella *)
				END_FOR

			ModBus.MB_Query.Read_StartAddress := 140 ;			(* richiedo lettura altri Parametri *)
			ModBus.MB_Query.Read_Quantity := 20;
			ModBus.MB_Start := TRUE;
			Read_StartAddress := 140 ;
			state := 37;
			END_IF
		END_IF

	37:	(* Risposta all'interrogazione *)
		IF NOT ModBus.MB_Start   THEN
			VerificaFuctionCode:=ModBus.MB_Resp.FunctionCode;
			VerificaNodoLetto:=ModBus.MB_Resp.SlaveAddress;

			IF ModBus.MB_MASTER.MB_Error<>0 THEN
				state := 300;
			ELSE

				FOR x:= 0 TO ModBus.MB_Query.Read_Quantity DO
					MB_RegistriLetti[Read_StartAddress+x ] := ModBus.MB_Resp.Data[x];   	(* Vedi tabella *)
				END_FOR

			ModBus.MB_Query.Read_StartAddress := 160 ;			(* richiedo lettura altri Parametri *)
			ModBus.MB_Query.Read_Quantity := 20;
			ModBus.MB_Start := TRUE;
			Read_StartAddress := 160 ;
			state := 38;
			END_IF
		END_IF

	38:	(* Risposta all'interrogazione *)
		IF NOT ModBus.MB_Start   THEN
			VerificaFuctionCode:=ModBus.MB_Resp.FunctionCode;
			VerificaNodoLetto:=ModBus.MB_Resp.SlaveAddress;

			IF ModBus.MB_MASTER.MB_Error<>0 THEN
				state := 300;
			ELSE

				FOR x:= 0 TO ModBus.MB_Query.Read_Quantity DO
					MB_RegistriLetti[Read_StartAddress+x ] := ModBus.MB_Resp.Data[x];   	(* Vedi tabella *)
				END_FOR

			ModBus.MB_Query.Read_StartAddress := 180 ;			(* richiedo lettura altri Parametri *)
			ModBus.MB_Query.Read_Quantity := 20;
			ModBus.MB_Start := TRUE;
			Read_StartAddress := 180 ;
			state := 39;
			END_IF
		END_IF

	39:	(* Risposta all'interrogazione *)
		IF NOT ModBus.MB_Start   THEN
			VerificaFuctionCode:=ModBus.MB_Resp.FunctionCode;
			VerificaNodoLetto:=ModBus.MB_Resp.SlaveAddress;

			IF ModBus.MB_MASTER.MB_Error<>0 THEN
				state := 300;
			ELSE

				FOR x:= 0 TO ModBus.MB_Query.Read_Quantity DO
					MB_RegistriLetti[Read_StartAddress+x ] := ModBus.MB_Resp.Data[x];   	(* Vedi tabella *)
				END_FOR

			ModBus.MB_Query.Read_StartAddress := 200 ;			(* richiedo lettura altri Parametri *)
			ModBus.MB_Query.Read_Quantity := 20;
			ModBus.MB_Start := TRUE;
			Read_StartAddress := 200 ;
			state := 40;
			END_IF
		END_IF

	40:	(* Risposta all'interrogazione *)
		IF NOT ModBus.MB_Start   THEN
			VerificaFuctionCode:=ModBus.MB_Resp.FunctionCode;
			VerificaNodoLetto:=ModBus.MB_Resp.SlaveAddress;

			IF ModBus.MB_MASTER.MB_Error<>0 THEN
				state := 300;
			ELSE

				FOR x:= 0 TO ModBus.MB_Query.Read_Quantity DO
					MB_RegistriLetti[Read_StartAddress+x ] := ModBus.MB_Resp.Data[x];   	(* Vedi tabella *)
				END_FOR

			ModBus.MB_Query.Read_StartAddress := 220 ;			(* richiedo lettura altri Parametri *)
			ModBus.MB_Query.Read_Quantity := 20;
			ModBus.MB_Start := TRUE;
			Read_StartAddress := 220 ;
			state := 41;
			END_IF
		END_IF

	41:	(* Risposta all'interrogazione *)
		IF NOT ModBus.MB_Start   THEN
			VerificaFuctionCode:=ModBus.MB_Resp.FunctionCode;
			VerificaNodoLetto:=ModBus.MB_Resp.SlaveAddress;

			IF ModBus.MB_MASTER.MB_Error<>0 THEN
				state := 300;
			ELSE

				FOR x:= 0 TO ModBus.MB_Query.Read_Quantity DO
					MB_RegistriLetti[Read_StartAddress+x ] := ModBus.MB_Resp.Data[x];   	(* Vedi tabella *)
				END_FOR

			ModBus.MB_Query.Read_StartAddress := 240 ;			(* richiedo lettura altri Parametri *)
			ModBus.MB_Query.Read_Quantity := 20;
			ModBus.MB_Start := TRUE;
			Read_StartAddress := 240 ;
			state := 42;
			END_IF
		END_IF

	42:	(* Risposta all'interrogazione *)
		IF NOT ModBus.MB_Start   THEN
			VerificaFuctionCode:=ModBus.MB_Resp.FunctionCode;
			VerificaNodoLetto:=ModBus.MB_Resp.SlaveAddress;

			IF ModBus.MB_MASTER.MB_Error<>0 THEN
				state := 300;
			ELSE

				FOR x:= 0 TO ModBus.MB_Query.Read_Quantity DO
					MB_RegistriLetti[Read_StartAddress+x ] := ModBus.MB_Resp.Data[x];   	(* Vedi tabella *)
				END_FOR

			ModBus.MB_Query.Read_StartAddress := 260 ;			(* richiedo lettura altri Parametri *)
			ModBus.MB_Query.Read_Quantity := 20;
			ModBus.MB_Start := TRUE;
			Read_StartAddress := 260 ;
			state := 43;
			END_IF
		END_IF

	43:	(* Risposta all'interrogazione *)
		IF NOT ModBus.MB_Start   THEN
			VerificaFuctionCode:=ModBus.MB_Resp.FunctionCode;
			VerificaNodoLetto:=ModBus.MB_Resp.SlaveAddress;

			IF ModBus.MB_MASTER.MB_Error<>0 THEN
				state := 300;
			ELSE

				FOR x:= 0 TO ModBus.MB_Query.Read_Quantity DO
					MB_RegistriLetti[Read_StartAddress+x ] := ModBus.MB_Resp.Data[x];   	(* Vedi tabella *)
				END_FOR

			ModBus.MB_Query.Read_StartAddress := 280 ;			(* richiedo lettura altri Parametri *)
			ModBus.MB_Query.Read_Quantity := 4;
			ModBus.MB_Start := TRUE;
			Read_StartAddress := 280 ;
			state := 44;
			END_IF
		END_IF

	44:	(* Risposta all'interrogazione *)
		IF NOT ModBus.MB_Start   THEN
			VerificaFuctionCode:=ModBus.MB_Resp.FunctionCode;
			VerificaNodoLetto:=ModBus.MB_Resp.SlaveAddress;

			IF ModBus.MB_MASTER.MB_Error<>0 THEN
				state := 300;
			ELSE

				FOR x:= 0 TO ModBus.MB_Query.Read_Quantity DO
					MB_RegistriLetti[Read_StartAddress+x ] := ModBus.MB_Resp.Data[x];   	(* Vedi tabella *)
				END_FOR

		(*	ModBus.MB_Query.Read_StartAddress := 280 ;			(* richiedo lettura altri Parametri *)
			ModBus.MB_Query.Read_Quantity := 4;
			ModBus.MB_Start := TRUE;
			Read_StartAddress := 280 ; *)
			state := 50;
			END_IF
		END_IF





	50:	(* Risposta all'interrogazione Holding*)

		Modbus.MB_Query.FunctionCode := 3;
		Read_StartAddress := 0 ;			(* richiedo lettura altri Parametri *)
		Read_Quantity := 20;
		ModBus.MB_Start := TRUE;
		state := 51;

	51:	(* Risposta all'interrogazione *)
		IF NOT ModBus.MB_Start   THEN
			VerificaFuctionCode:=ModBus.MB_Resp.FunctionCode;
			VerificaNodoLetto:=ModBus.MB_Resp.SlaveAddress;

			IF ModBus.MB_MASTER.MB_Error<>0 THEN
				state := 300;
			ELSE

				FOR x:= 0 TO ModBus.MB_Query.Read_Quantity DO
					MB_RegistriHoldingLetti[Read_StartAddress+x ] := ModBus.MB_Resp.Data[x];   	(* Vedi tabella *)
				END_FOR

			ModBus.MB_Query.Read_StartAddress := 0 ;			(* richiedo lettura altri Parametri *)
			ModBus.MB_Query.Read_Quantity := 20;
			ModBus.MB_Start := TRUE;
			Read_StartAddress := 0 ;
			state := 511;
			END_IF
		END_IF


	511:	(* Risposta all'interrogazione *)
		IF NOT ModBus.MB_Start   THEN
			VerificaFuctionCode:=ModBus.MB_Resp.FunctionCode;
			VerificaNodoLetto:=ModBus.MB_Resp.SlaveAddress;

			IF ModBus.MB_MASTER.MB_Error<>0 THEN
				state := 300;
			ELSE

				FOR x:= 0 TO ModBus.MB_Query.Read_Quantity DO
					MB_RegistriHoldingLetti[Read_StartAddress+x ] := ModBus.MB_Resp.Data[x];   	(* Vedi tabella *)
				END_FOR

			ModBus.MB_Query.Read_StartAddress := 20 ;			(* richiedo lettura altri Parametri *)
			ModBus.MB_Query.Read_Quantity := 20;
			ModBus.MB_Start := TRUE;
			Read_StartAddress := 20 ;
			state := 52;
			END_IF
		END_IF

	52:	(* Risposta all'interrogazione *)
		IF NOT ModBus.MB_Start   THEN
			VerificaFuctionCode:=ModBus.MB_Resp.FunctionCode;
			VerificaNodoLetto:=ModBus.MB_Resp.SlaveAddress;

			IF ModBus.MB_MASTER.MB_Error<>0 THEN
				state := 300;
			ELSE

				FOR x:= 0 TO ModBus.MB_Query.Read_Quantity DO
					MB_RegistriHoldingLetti[Read_StartAddress+x ] := ModBus.MB_Resp.Data[x];   	(* Vedi tabella *)
				END_FOR

			ModBus.MB_Query.Read_StartAddress := 40 ;			(* richiedo lettura altri Parametri *)
			ModBus.MB_Query.Read_Quantity := 20;
			ModBus.MB_Start := TRUE;
			Read_StartAddress := 40 ;
			state := 53;
			END_IF
		END_IF

	53:	(* Risposta all'interrogazione *)
		IF NOT ModBus.MB_Start   THEN
			VerificaFuctionCode:=ModBus.MB_Resp.FunctionCode;
			VerificaNodoLetto:=ModBus.MB_Resp.SlaveAddress;

			IF ModBus.MB_MASTER.MB_Error<>0 THEN
				state := 300;
			ELSE

				FOR x:= 0 TO ModBus.MB_Query.Read_Quantity DO
					MB_RegistriHoldingLetti[Read_StartAddress+x ] := ModBus.MB_Resp.Data[x];   	(* Vedi tabella *)
				END_FOR

			ModBus.MB_Query.Read_StartAddress := 60 ;			(* richiedo lettura altri Parametri *)
			ModBus.MB_Query.Read_Quantity := 20;
			ModBus.MB_Start := TRUE;
			Read_StartAddress := 60 ;
			state := 54;
			END_IF
		END_IF

	54:	(* Risposta all'interrogazione *)
		IF NOT ModBus.MB_Start   THEN
			VerificaFuctionCode:=ModBus.MB_Resp.FunctionCode;
			VerificaNodoLetto:=ModBus.MB_Resp.SlaveAddress;

			IF ModBus.MB_MASTER.MB_Error<>0 THEN
				state := 300;
			ELSE

				FOR x:= 0 TO ModBus.MB_Query.Read_Quantity DO
					MB_RegistriHoldingLetti[Read_StartAddress+x ] := ModBus.MB_Resp.Data[x];   	(* Vedi tabella *)
				END_FOR

			ModBus.MB_Query.Read_StartAddress := 80 ;			(* richiedo lettura altri Parametri *)
			ModBus.MB_Query.Read_Quantity := 20;
			ModBus.MB_Start := TRUE;
			Read_StartAddress := 80 ;
			state := 55;
			END_IF
		END_IF

	55:	(* Risposta all'interrogazione *)
		IF NOT ModBus.MB_Start   THEN
			VerificaFuctionCode:=ModBus.MB_Resp.FunctionCode;
			VerificaNodoLetto:=ModBus.MB_Resp.SlaveAddress;

			IF ModBus.MB_MASTER.MB_Error<>0 THEN
				state := 300;
			ELSE

				FOR x:= 0 TO ModBus.MB_Query.Read_Quantity DO
					MB_RegistriHoldingLetti[Read_StartAddress+x ] := ModBus.MB_Resp.Data[x];   	(* Vedi tabella *)
				END_FOR

			ModBus.MB_Query.Read_StartAddress := 100 ;			(* richiedo lettura altri Parametri *)
			ModBus.MB_Query.Read_Quantity := 20;
			ModBus.MB_Start := TRUE;
			Read_StartAddress := 100 ;
			state := 56;
			END_IF
		END_IF

	56:	(* Risposta all'interrogazione *)
		IF NOT ModBus.MB_Start   THEN
			VerificaFuctionCode:=ModBus.MB_Resp.FunctionCode;
			VerificaNodoLetto:=ModBus.MB_Resp.SlaveAddress;

			IF ModBus.MB_MASTER.MB_Error<>0 THEN
				state := 300;
			ELSE

				FOR x:= 0 TO ModBus.MB_Query.Read_Quantity DO
					MB_RegistriHoldingLetti[Read_StartAddress+x ] := ModBus.MB_Resp.Data[x];   	(* Vedi tabella *)
				END_FOR

			ModBus.MB_Query.Read_StartAddress := 120 ;			(* richiedo lettura altri Parametri *)
			ModBus.MB_Query.Read_Quantity := 20;
			ModBus.MB_Start := TRUE;
			Read_StartAddress := 120 ;
			state := 57;
			END_IF
		END_IF

	57:	(* Risposta all'interrogazione *)
		IF NOT ModBus.MB_Start   THEN
			VerificaFuctionCode:=ModBus.MB_Resp.FunctionCode;
			VerificaNodoLetto:=ModBus.MB_Resp.SlaveAddress;

			IF ModBus.MB_MASTER.MB_Error<>0 THEN
				state := 300;
			ELSE

				FOR x:= 0 TO ModBus.MB_Query.Read_Quantity DO
					MB_RegistriHoldingLetti[Read_StartAddress+x ] := ModBus.MB_Resp.Data[x];   	(* Vedi tabella *)
				END_FOR

			ModBus.MB_Query.Read_StartAddress := 140 ;			(* richiedo lettura altri Parametri *)
			ModBus.MB_Query.Read_Quantity := 20;
			ModBus.MB_Start := TRUE;
			Read_StartAddress := 140 ;
			state := 58;
			END_IF
		END_IF

	58:	(* Risposta all'interrogazione *)
		IF NOT ModBus.MB_Start   THEN
			VerificaFuctionCode:=ModBus.MB_Resp.FunctionCode;
			VerificaNodoLetto:=ModBus.MB_Resp.SlaveAddress;

			IF ModBus.MB_MASTER.MB_Error<>0 THEN
				state := 300;
			ELSE

				FOR x:= 0 TO ModBus.MB_Query.Read_Quantity DO
					MB_RegistriHoldingLetti[Read_StartAddress+x ] := ModBus.MB_Resp.Data[x];   	(* Vedi tabella *)
				END_FOR

			ModBus.MB_Query.Read_StartAddress := 160 ;			(* richiedo lettura altri Parametri *)
			ModBus.MB_Query.Read_Quantity := 8;
			ModBus.MB_Start := TRUE;
			Read_StartAddress := 160 ;
			state := 59;
			END_IF
		END_IF

	59:	(* Risposta all'interrogazione *)
		IF NOT ModBus.MB_Start   THEN
			VerificaFuctionCode:=ModBus.MB_Resp.FunctionCode;
			VerificaNodoLetto:=ModBus.MB_Resp.SlaveAddress;

			IF ModBus.MB_MASTER.MB_Error<>0 THEN
				state := 300;
			ELSE

				FOR x:= 0 TO ModBus.MB_Query.Read_Quantity DO
					MB_RegistriHoldingLetti[Read_StartAddress+x ] := ModBus.MB_Resp.Data[x];   	(* Vedi tabella *)
				END_FOR

		(*	ModBus.MB_Query.Read_StartAddress := 160 ;			(* richiedo lettura altri Parametri *)
			ModBus.MB_Query.Read_Quantity := 20;
			ModBus.MB_Start := TRUE;
			Read_StartAddress := 160 ; *)
			state := 100;
			END_IF
		END_IF





	100: (* Rispota Altri paramenti Digital Input *)
		IF NOT ModBus.MB_Start  THEN

			IF ModBus.MB_MASTER.MB_Error<>0 THEN
				state := 300;
			ELSE
				Modbus.MB_Query.SlaveAddress := Address;
				Modbus.MB_Query.FunctionCode := 2;
				ModBus.MB_Query.Read_StartAddress := 0;	(* richiedo lettura altri Parametri *)
				ModBus.MB_Query.Read_Quantity := 64;
				ModBus.MB_Start := TRUE;

				state:=105;
			END_IF
		END_IF
	105: (* Rispota Altri paramenti *)

		IF NOT ModBus.MB_Start  THEN

			IF ModBus.MB_MASTER.MB_Error<>0 THEN
				state := 300;
			ELSE

				MB_BitStato[0]:=ModBus.MB_MASTER.ReceiveBuffer.Data[3].0; (*Vedi Tabella *)
				MB_BitStato[1]:=ModBus.MB_MASTER.ReceiveBuffer.Data[3].1; (*Vedi Tabella *)
				MB_BitStato[2]:=ModBus.MB_MASTER.ReceiveBuffer.Data[3].2; (*Vedi Tabella *)
				MB_BitStato[3]:=ModBus.MB_MASTER.ReceiveBuffer.Data[3].3; (*Vedi Tabella *)
				MB_BitStato[4]:=ModBus.MB_MASTER.ReceiveBuffer.Data[3].4; (*Vedi Tabella *)
				MB_BitStato[5]:=ModBus.MB_MASTER.ReceiveBuffer.Data[3].5; (*Vedi Tabella *)
				MB_BitStato[6]:=ModBus.MB_MASTER.ReceiveBuffer.Data[3].6; (*Vedi Tabella *)
				MB_BitStato[7]:=ModBus.MB_MASTER.ReceiveBuffer.Data[3].7; (*Vedi Tabella *)
				MB_BitStato[8]:=ModBus.MB_MASTER.ReceiveBuffer.Data[4].0; (*Vedi Tabella *)
				MB_BitStato[9]:=ModBus.MB_MASTER.ReceiveBuffer.Data[4].1; (*Vedi Tabella *)
				MB_BitStato[10]:=ModBus.MB_MASTER.ReceiveBuffer.Data[4].2; (*Vedi Tabella *)
				MB_BitStato[11]:=ModBus.MB_MASTER.ReceiveBuffer.Data[4].3; (*Vedi Tabella *)
				MB_BitStato[12]:=ModBus.MB_MASTER.ReceiveBuffer.Data[4].4; (*Vedi Tabella *)
				MB_BitStato[13]:=ModBus.MB_MASTER.ReceiveBuffer.Data[4].5; (*Vedi Tabella *)
				MB_BitStato[14]:=ModBus.MB_MASTER.ReceiveBuffer.Data[4].6; (*Vedi Tabella *)
				MB_BitStato[15]:=ModBus.MB_MASTER.ReceiveBuffer.Data[4].7; (*Vedi Tabella *)
				MB_BitStato[16]:=ModBus.MB_MASTER.ReceiveBuffer.Data[5].0; (*Vedi Tabella *)
				MB_BitStato[17]:=ModBus.MB_MASTER.ReceiveBuffer.Data[5].1; (*Vedi Tabella *)
				MB_BitStato[18]:=ModBus.MB_MASTER.ReceiveBuffer.Data[5].2; (*Vedi Tabella *)
				MB_BitStato[19]:=ModBus.MB_MASTER.ReceiveBuffer.Data[5].3; (*Vedi Tabella *)
				MB_BitStato[20]:=ModBus.MB_MASTER.ReceiveBuffer.Data[5].4; (*Vedi Tabella *)
				MB_BitStato[21]:=ModBus.MB_MASTER.ReceiveBuffer.Data[5].5; (*Vedi Tabella *)
				MB_BitStato[22]:=ModBus.MB_MASTER.ReceiveBuffer.Data[5].6; (*Vedi Tabella *)
				MB_BitStato[23]:=ModBus.MB_MASTER.ReceiveBuffer.Data[5].7; (*Vedi Tabella *)
				MB_BitStato[24]:=ModBus.MB_MASTER.ReceiveBuffer.Data[6].0; (*Vedi Tabella *)
				MB_BitStato[25]:=ModBus.MB_MASTER.ReceiveBuffer.Data[6].1; (*Vedi Tabella *)
				MB_BitStato[26]:=ModBus.MB_MASTER.ReceiveBuffer.Data[6].2; (*Vedi Tabella *)
				MB_BitStato[27]:=ModBus.MB_MASTER.ReceiveBuffer.Data[6].3; (*Vedi Tabella *)
				MB_BitStato[28]:=ModBus.MB_MASTER.ReceiveBuffer.Data[6].4; (*Vedi Tabella *)
				MB_BitStato[29]:=ModBus.MB_MASTER.ReceiveBuffer.Data[6].5; (*Vedi Tabella *)
				MB_BitStato[30]:=ModBus.MB_MASTER.ReceiveBuffer.Data[6].6; (*Vedi Tabella *)
				MB_BitStato[31]:=ModBus.MB_MASTER.ReceiveBuffer.Data[6].7; (*Vedi Tabella *)
				MB_BitStato[32]:=ModBus.MB_MASTER.ReceiveBuffer.Data[7].0; (*Vedi Tabella *)
				MB_BitStato[33]:=ModBus.MB_MASTER.ReceiveBuffer.Data[7].1; (*Vedi Tabella *)
				MB_BitStato[34]:=ModBus.MB_MASTER.ReceiveBuffer.Data[7].2; (*Vedi Tabella *)
				MB_BitStato[35]:=ModBus.MB_MASTER.ReceiveBuffer.Data[7].3; (*Vedi Tabella *)
				MB_BitStato[36]:=ModBus.MB_MASTER.ReceiveBuffer.Data[7].4; (*Vedi Tabella *)
				MB_BitStato[37]:=ModBus.MB_MASTER.ReceiveBuffer.Data[7].5; (*Vedi Tabella *)
				MB_BitStato[38]:=ModBus.MB_MASTER.ReceiveBuffer.Data[7].6; (*Vedi Tabella *)
				MB_BitStato[39]:=ModBus.MB_MASTER.ReceiveBuffer.Data[7].7; (*Vedi Tabella *)
				MB_BitStato[40]:=ModBus.MB_MASTER.ReceiveBuffer.Data[8].0; (*Vedi Tabella *)
				MB_BitStato[41]:=ModBus.MB_MASTER.ReceiveBuffer.Data[8].1; (*Vedi Tabella *)
				MB_BitStato[42]:=ModBus.MB_MASTER.ReceiveBuffer.Data[8].2; (*Vedi Tabella *)
				MB_BitStato[43]:=ModBus.MB_MASTER.ReceiveBuffer.Data[8].3; (*Vedi Tabella *)
				MB_BitStato[44]:=ModBus.MB_MASTER.ReceiveBuffer.Data[8].4; (*Vedi Tabella *)
				MB_BitStato[45]:=ModBus.MB_MASTER.ReceiveBuffer.Data[8].5; (*Vedi Tabella *)
				MB_BitStato[46]:=ModBus.MB_MASTER.ReceiveBuffer.Data[8].6; (*Vedi Tabella *)
				MB_BitStato[47]:=ModBus.MB_MASTER.ReceiveBuffer.Data[8].7; (*Vedi Tabella *)
				MB_BitStato[48]:=ModBus.MB_MASTER.ReceiveBuffer.Data[9].0; (*Vedi Tabella *)
				MB_BitStato[49]:=ModBus.MB_MASTER.ReceiveBuffer.Data[9].1; (*Vedi Tabella *)
				MB_BitStato[50]:=ModBus.MB_MASTER.ReceiveBuffer.Data[9].2; (*Vedi Tabella *)
				MB_BitStato[51]:=ModBus.MB_MASTER.ReceiveBuffer.Data[9].3; (*Vedi Tabella *)
				MB_BitStato[52]:=ModBus.MB_MASTER.ReceiveBuffer.Data[9].4; (*Vedi Tabella *)
				MB_BitStato[53]:=ModBus.MB_MASTER.ReceiveBuffer.Data[9].5; (*Vedi Tabella *)
				MB_BitStato[54]:=ModBus.MB_MASTER.ReceiveBuffer.Data[9].6; (*Vedi Tabella *)
				MB_BitStato[55]:=ModBus.MB_MASTER.ReceiveBuffer.Data[9].7; (*Vedi Tabella *)
				MB_BitStato[56]:=ModBus.MB_MASTER.ReceiveBuffer.Data[10].0; (*Vedi Tabella *)
				MB_BitStato[57]:=ModBus.MB_MASTER.ReceiveBuffer.Data[10].1; (*Vedi Tabella *)
				MB_BitStato[58]:=ModBus.MB_MASTER.ReceiveBuffer.Data[10].2; (*Vedi Tabella *)
				MB_BitStato[59]:=ModBus.MB_MASTER.ReceiveBuffer.Data[10].3; (*Vedi Tabella *)
				MB_BitStato[60]:=ModBus.MB_MASTER.ReceiveBuffer.Data[10].4; (*Vedi Tabella *)
				MB_BitStato[61]:=ModBus.MB_MASTER.ReceiveBuffer.Data[10].5; (*Vedi Tabella *)
				MB_BitStato[62]:=ModBus.MB_MASTER.ReceiveBuffer.Data[10].6; (*Vedi Tabella *)
				MB_BitStato[63]:=ModBus.MB_MASTER.ReceiveBuffer.Data[10].7; (*Vedi Tabella *)

				state:=110;

			END_IF
		END_IF

	110: (* Rispota Altri paramenti *)
		IF NOT ModBus.MB_Start  THEN

			IF ModBus.MB_MASTER.MB_Error<>0 THEN
				state := 300;
			ELSE
				Modbus.MB_Query.SlaveAddress := Address;
				Modbus.MB_Query.FunctionCode := 2;
				ModBus.MB_Query.Read_StartAddress := 64;
				ModBus.MB_Query.Read_Quantity := 64;
				ModBus.MB_Start := TRUE;

				state:=115;
			END_IF
		END_IF
	115: (* Rispota Altri paramenti *)

		IF NOT ModBus.MB_Start  THEN

			IF ModBus.MB_MASTER.MB_Error<>0 THEN
				state := 300;
			ELSE

				MB_BitStato[64]:=ModBus.MB_MASTER.ReceiveBuffer.Data[3].0; (*Vedi Tabella *)
				MB_BitStato[65]:=ModBus.MB_MASTER.ReceiveBuffer.Data[3].1; (*Vedi Tabella *)
				MB_BitStato[66]:=ModBus.MB_MASTER.ReceiveBuffer.Data[3].2; (*Vedi Tabella *)
				MB_BitStato[67]:=ModBus.MB_MASTER.ReceiveBuffer.Data[3].3; (*Vedi Tabella *)
				MB_BitStato[68]:=ModBus.MB_MASTER.ReceiveBuffer.Data[3].4; (*Vedi Tabella *)
				MB_BitStato[69]:=ModBus.MB_MASTER.ReceiveBuffer.Data[3].5; (*Vedi Tabella *)
				MB_BitStato[70]:=ModBus.MB_MASTER.ReceiveBuffer.Data[3].6; (*Vedi Tabella *)
				MB_BitStato[71]:=ModBus.MB_MASTER.ReceiveBuffer.Data[3].7; (*Vedi Tabella *)
				MB_BitStato[72]:=ModBus.MB_MASTER.ReceiveBuffer.Data[4].0; (*Vedi Tabella *)
				MB_BitStato[73]:=ModBus.MB_MASTER.ReceiveBuffer.Data[4].1; (*Vedi Tabella *)
				MB_BitStato[74]:=ModBus.MB_MASTER.ReceiveBuffer.Data[4].2; (*Vedi Tabella *)
				MB_BitStato[75]:=ModBus.MB_MASTER.ReceiveBuffer.Data[4].3; (*Vedi Tabella *)
				MB_BitStato[76]:=ModBus.MB_MASTER.ReceiveBuffer.Data[4].4; (*Vedi Tabella *)
				MB_BitStato[77]:=ModBus.MB_MASTER.ReceiveBuffer.Data[4].5; (*Vedi Tabella *)
				MB_BitStato[78]:=ModBus.MB_MASTER.ReceiveBuffer.Data[4].6; (*Vedi Tabella *)
				MB_BitStato[79]:=ModBus.MB_MASTER.ReceiveBuffer.Data[4].7; (*Vedi Tabella *)
				MB_BitStato[80]:=ModBus.MB_MASTER.ReceiveBuffer.Data[5].0; (*Vedi Tabella *)
				MB_BitStato[81]:=ModBus.MB_MASTER.ReceiveBuffer.Data[5].1; (*Vedi Tabella *)
				MB_BitStato[82]:=ModBus.MB_MASTER.ReceiveBuffer.Data[5].2; (*Vedi Tabella *)
				MB_BitStato[83]:=ModBus.MB_MASTER.ReceiveBuffer.Data[5].3; (*Vedi Tabella *)
				MB_BitStato[84]:=ModBus.MB_MASTER.ReceiveBuffer.Data[5].4; (*Vedi Tabella *)
				MB_BitStato[85]:=ModBus.MB_MASTER.ReceiveBuffer.Data[5].5; (*Vedi Tabella *)
				MB_BitStato[86]:=ModBus.MB_MASTER.ReceiveBuffer.Data[5].6; (*Vedi Tabella *)
				MB_BitStato[87]:=ModBus.MB_MASTER.ReceiveBuffer.Data[5].7; (*Vedi Tabella *)
				MB_BitStato[88]:=ModBus.MB_MASTER.ReceiveBuffer.Data[6].0; (*Vedi Tabella *)
				MB_BitStato[89]:=ModBus.MB_MASTER.ReceiveBuffer.Data[6].1; (*Vedi Tabella *)
				MB_BitStato[90]:=ModBus.MB_MASTER.ReceiveBuffer.Data[6].2; (*Vedi Tabella *)
				MB_BitStato[91]:=ModBus.MB_MASTER.ReceiveBuffer.Data[6].3; (*Vedi Tabella *)
				MB_BitStato[92]:=ModBus.MB_MASTER.ReceiveBuffer.Data[6].4; (*Vedi Tabella *)
				MB_BitStato[93]:=ModBus.MB_MASTER.ReceiveBuffer.Data[6].5; (*Vedi Tabella *)
				MB_BitStato[94]:=ModBus.MB_MASTER.ReceiveBuffer.Data[6].6; (*Vedi Tabella *)
				MB_BitStato[95]:=ModBus.MB_MASTER.ReceiveBuffer.Data[6].7; (*Vedi Tabella *)
				MB_BitStato[96]:=ModBus.MB_MASTER.ReceiveBuffer.Data[7].0; (*Vedi Tabella *)
				MB_BitStato[97]:=ModBus.MB_MASTER.ReceiveBuffer.Data[7].1; (*Vedi Tabella *)
				MB_BitStato[98]:=ModBus.MB_MASTER.ReceiveBuffer.Data[7].2; (*Vedi Tabella *)
				MB_BitStato[99]:=ModBus.MB_MASTER.ReceiveBuffer.Data[7].3; (*Vedi Tabella *)
				MB_BitStato[100]:=ModBus.MB_MASTER.ReceiveBuffer.Data[7].4; (*Vedi Tabella *)
				MB_BitStato[101]:=ModBus.MB_MASTER.ReceiveBuffer.Data[7].5; (*Vedi Tabella *)
				MB_BitStato[102]:=ModBus.MB_MASTER.ReceiveBuffer.Data[7].6; (*Vedi Tabella *)
				MB_BitStato[103]:=ModBus.MB_MASTER.ReceiveBuffer.Data[7].7; (*Vedi Tabella *)
				MB_BitStato[104]:=ModBus.MB_MASTER.ReceiveBuffer.Data[8].0; (*Vedi Tabella *)
				MB_BitStato[105]:=ModBus.MB_MASTER.ReceiveBuffer.Data[8].1; (*Vedi Tabella *)
				MB_BitStato[106]:=ModBus.MB_MASTER.ReceiveBuffer.Data[8].2; (*Vedi Tabella *)
				MB_BitStato[107]:=ModBus.MB_MASTER.ReceiveBuffer.Data[8].3; (*Vedi Tabella *)
				MB_BitStato[108]:=ModBus.MB_MASTER.ReceiveBuffer.Data[8].4; (*Vedi Tabella *)
				MB_BitStato[109]:=ModBus.MB_MASTER.ReceiveBuffer.Data[8].5; (*Vedi Tabella *)
				MB_BitStato[110]:=ModBus.MB_MASTER.ReceiveBuffer.Data[8].6; (*Vedi Tabella *)
				MB_BitStato[111]:=ModBus.MB_MASTER.ReceiveBuffer.Data[8].7; (*Vedi Tabella *)
				MB_BitStato[112]:=ModBus.MB_MASTER.ReceiveBuffer.Data[9].0; (*Vedi Tabella *)
				MB_BitStato[113]:=ModBus.MB_MASTER.ReceiveBuffer.Data[9].1; (*Vedi Tabella *)
				MB_BitStato[114]:=ModBus.MB_MASTER.ReceiveBuffer.Data[9].2; (*Vedi Tabella *)
				MB_BitStato[115]:=ModBus.MB_MASTER.ReceiveBuffer.Data[9].3; (*Vedi Tabella *)
				MB_BitStato[116]:=ModBus.MB_MASTER.ReceiveBuffer.Data[9].4; (*Vedi Tabella *)
				MB_BitStato[117]:=ModBus.MB_MASTER.ReceiveBuffer.Data[9].5; (*Vedi Tabella *)
				MB_BitStato[118]:=ModBus.MB_MASTER.ReceiveBuffer.Data[9].6; (*Vedi Tabella *)
				MB_BitStato[119]:=ModBus.MB_MASTER.ReceiveBuffer.Data[9].7; (*Vedi Tabella *)
				MB_BitStato[120]:=ModBus.MB_MASTER.ReceiveBuffer.Data[10].0; (*Vedi Tabella *)
				MB_BitStato[121]:=ModBus.MB_MASTER.ReceiveBuffer.Data[10].1; (*Vedi Tabella *)
				MB_BitStato[122]:=ModBus.MB_MASTER.ReceiveBuffer.Data[10].2; (*Vedi Tabella *)
				MB_BitStato[123]:=ModBus.MB_MASTER.ReceiveBuffer.Data[10].3; (*Vedi Tabella *)
				MB_BitStato[124]:=ModBus.MB_MASTER.ReceiveBuffer.Data[10].4; (*Vedi Tabella *)
				MB_BitStato[125]:=ModBus.MB_MASTER.ReceiveBuffer.Data[10].5; (*Vedi Tabella *)
				MB_BitStato[126]:=ModBus.MB_MASTER.ReceiveBuffer.Data[10].6; (*Vedi Tabella *)
				MB_BitStato[127]:=ModBus.MB_MASTER.ReceiveBuffer.Data[10].7; (*Vedi Tabella *)


				state:=120;

			END_IF
		END_IF


	120: (* Rispota Altri paramenti *)
		IF NOT ModBus.MB_Start  THEN

			IF ModBus.MB_MASTER.MB_Error<>0 THEN
				state := 300;
			ELSE
				Modbus.MB_Query.SlaveAddress := Address;
				Modbus.MB_Query.FunctionCode := 2;
				ModBus.MB_Query.Read_StartAddress := 128;
				ModBus.MB_Query.Read_Quantity := 64;
				ModBus.MB_Start := TRUE;

				state:=125;
			END_IF
		END_IF
	125: (* Rispota Altri paramenti *)

		IF NOT ModBus.MB_Start  THEN

			IF ModBus.MB_MASTER.MB_Error<>0 THEN
				state := 300;
			ELSE

				MB_BitStato[128]:=ModBus.MB_MASTER.ReceiveBuffer.Data[3].0; (*Vedi Tabella *)
				MB_BitStato[129]:=ModBus.MB_MASTER.ReceiveBuffer.Data[3].1; (*Vedi Tabella *)
				MB_BitStato[130]:=ModBus.MB_MASTER.ReceiveBuffer.Data[3].2; (*Vedi Tabella *)
				MB_BitStato[131]:=ModBus.MB_MASTER.ReceiveBuffer.Data[3].3; (*Vedi Tabella *)
				MB_BitStato[132]:=ModBus.MB_MASTER.ReceiveBuffer.Data[3].4; (*Vedi Tabella *)
				MB_BitStato[133]:=ModBus.MB_MASTER.ReceiveBuffer.Data[3].5; (*Vedi Tabella *)
				MB_BitStato[134]:=ModBus.MB_MASTER.ReceiveBuffer.Data[3].6; (*Vedi Tabella *)
				MB_BitStato[135]:=ModBus.MB_MASTER.ReceiveBuffer.Data[3].7; (*Vedi Tabella *)
				MB_BitStato[136]:=ModBus.MB_MASTER.ReceiveBuffer.Data[4].0; (*Vedi Tabella *)
				MB_BitStato[137]:=ModBus.MB_MASTER.ReceiveBuffer.Data[4].1; (*Vedi Tabella *)
				MB_BitStato[138]:=ModBus.MB_MASTER.ReceiveBuffer.Data[4].2; (*Vedi Tabella *)
				MB_BitStato[139]:=ModBus.MB_MASTER.ReceiveBuffer.Data[4].3; (*Vedi Tabella *)
				MB_BitStato[140]:=ModBus.MB_MASTER.ReceiveBuffer.Data[4].4; (*Vedi Tabella *)
				MB_BitStato[141]:=ModBus.MB_MASTER.ReceiveBuffer.Data[4].5; (*Vedi Tabella *)
				MB_BitStato[142]:=ModBus.MB_MASTER.ReceiveBuffer.Data[4].6; (*Vedi Tabella *)
				MB_BitStato[143]:=ModBus.MB_MASTER.ReceiveBuffer.Data[4].7; (*Vedi Tabella *)
				MB_BitStato[144]:=ModBus.MB_MASTER.ReceiveBuffer.Data[5].0; (*Vedi Tabella *)
				MB_BitStato[145]:=ModBus.MB_MASTER.ReceiveBuffer.Data[5].1; (*Vedi Tabella *)
				MB_BitStato[146]:=ModBus.MB_MASTER.ReceiveBuffer.Data[5].2; (*Vedi Tabella *)
				MB_BitStato[147]:=ModBus.MB_MASTER.ReceiveBuffer.Data[5].3; (*Vedi Tabella *)
				MB_BitStato[148]:=ModBus.MB_MASTER.ReceiveBuffer.Data[5].4; (*Vedi Tabella *)
				MB_BitStato[149]:=ModBus.MB_MASTER.ReceiveBuffer.Data[5].5; (*Vedi Tabella *)
				MB_BitStato[150]:=ModBus.MB_MASTER.ReceiveBuffer.Data[5].6; (*Vedi Tabella *)
				MB_BitStato[151]:=ModBus.MB_MASTER.ReceiveBuffer.Data[5].7; (*Vedi Tabella *)
				MB_BitStato[152]:=ModBus.MB_MASTER.ReceiveBuffer.Data[6].0; (*Vedi Tabella *)
				MB_BitStato[153]:=ModBus.MB_MASTER.ReceiveBuffer.Data[6].1; (*Vedi Tabella *)
				MB_BitStato[154]:=ModBus.MB_MASTER.ReceiveBuffer.Data[6].2; (*Vedi Tabella *)
				MB_BitStato[155]:=ModBus.MB_MASTER.ReceiveBuffer.Data[6].3; (*Vedi Tabella *)
				MB_BitStato[156]:=ModBus.MB_MASTER.ReceiveBuffer.Data[6].4; (*Vedi Tabella *)
				MB_BitStato[157]:=ModBus.MB_MASTER.ReceiveBuffer.Data[6].5; (*Vedi Tabella *)
				MB_BitStato[158]:=ModBus.MB_MASTER.ReceiveBuffer.Data[6].6; (*Vedi Tabella *)
				MB_BitStato[159]:=ModBus.MB_MASTER.ReceiveBuffer.Data[6].7; (*Vedi Tabella *)
				MB_BitStato[160]:=ModBus.MB_MASTER.ReceiveBuffer.Data[7].0; (*Vedi Tabella *)
				MB_BitStato[161]:=ModBus.MB_MASTER.ReceiveBuffer.Data[7].1; (*Vedi Tabella *)
				MB_BitStato[162]:=ModBus.MB_MASTER.ReceiveBuffer.Data[7].2; (*Vedi Tabella *)
				MB_BitStato[163]:=ModBus.MB_MASTER.ReceiveBuffer.Data[7].3; (*Vedi Tabella *)
				MB_BitStato[164]:=ModBus.MB_MASTER.ReceiveBuffer.Data[7].4; (*Vedi Tabella *)
				MB_BitStato[165]:=ModBus.MB_MASTER.ReceiveBuffer.Data[7].5; (*Vedi Tabella *)
				MB_BitStato[166]:=ModBus.MB_MASTER.ReceiveBuffer.Data[7].6; (*Vedi Tabella *)
				MB_BitStato[167]:=ModBus.MB_MASTER.ReceiveBuffer.Data[7].7; (*Vedi Tabella *)
				MB_BitStato[168]:=ModBus.MB_MASTER.ReceiveBuffer.Data[8].0; (*Vedi Tabella *)
				MB_BitStato[169]:=ModBus.MB_MASTER.ReceiveBuffer.Data[8].1; (*Vedi Tabella *)
				MB_BitStato[170]:=ModBus.MB_MASTER.ReceiveBuffer.Data[8].2; (*Vedi Tabella *)
				MB_BitStato[171]:=ModBus.MB_MASTER.ReceiveBuffer.Data[8].3; (*Vedi Tabella *)
				MB_BitStato[172]:=ModBus.MB_MASTER.ReceiveBuffer.Data[8].4; (*Vedi Tabella *)
				MB_BitStato[173]:=ModBus.MB_MASTER.ReceiveBuffer.Data[8].5; (*Vedi Tabella *)
				MB_BitStato[174]:=ModBus.MB_MASTER.ReceiveBuffer.Data[8].6; (*Vedi Tabella *)
				MB_BitStato[175]:=ModBus.MB_MASTER.ReceiveBuffer.Data[8].7; (*Vedi Tabella *)
				MB_BitStato[176]:=ModBus.MB_MASTER.ReceiveBuffer.Data[9].0; (*Vedi Tabella *)
				MB_BitStato[177]:=ModBus.MB_MASTER.ReceiveBuffer.Data[9].1; (*Vedi Tabella *)
				MB_BitStato[178]:=ModBus.MB_MASTER.ReceiveBuffer.Data[9].2; (*Vedi Tabella *)
				MB_BitStato[179]:=ModBus.MB_MASTER.ReceiveBuffer.Data[9].3; (*Vedi Tabella *)
				MB_BitStato[180]:=ModBus.MB_MASTER.ReceiveBuffer.Data[9].4; (*Vedi Tabella *)
				MB_BitStato[181]:=ModBus.MB_MASTER.ReceiveBuffer.Data[9].5; (*Vedi Tabella *)
				MB_BitStato[182]:=ModBus.MB_MASTER.ReceiveBuffer.Data[9].6; (*Vedi Tabella *)
				MB_BitStato[183]:=ModBus.MB_MASTER.ReceiveBuffer.Data[9].7; (*Vedi Tabella *)
				MB_BitStato[184]:=ModBus.MB_MASTER.ReceiveBuffer.Data[10].0; (*Vedi Tabella *)
				MB_BitStato[185]:=ModBus.MB_MASTER.ReceiveBuffer.Data[10].1; (*Vedi Tabella *)
				MB_BitStato[186]:=ModBus.MB_MASTER.ReceiveBuffer.Data[10].2; (*Vedi Tabella *)
				MB_BitStato[187]:=ModBus.MB_MASTER.ReceiveBuffer.Data[10].3; (*Vedi Tabella *)
				MB_BitStato[188]:=ModBus.MB_MASTER.ReceiveBuffer.Data[10].4; (*Vedi Tabella *)
				MB_BitStato[189]:=ModBus.MB_MASTER.ReceiveBuffer.Data[10].5; (*Vedi Tabella *)
				MB_BitStato[190]:=ModBus.MB_MASTER.ReceiveBuffer.Data[10].6; (*Vedi Tabella *)
				MB_BitStato[191]:=ModBus.MB_MASTER.ReceiveBuffer.Data[10].7; (*Vedi Tabella *)


				state:=130;

			END_IF
		END_IF


	130: (* Rispota Altri paramenti COIL *)
		IF NOT ModBus.MB_Start  THEN

			IF ModBus.MB_MASTER.MB_Error<>0 THEN
				state := 300;
			ELSE
				Modbus.MB_Query.SlaveAddress := Address;
				Modbus.MB_Query.FunctionCode := 2;
				ModBus.MB_Query.Read_StartAddress := 192;	(* richiedo lettura altri Parametri *)
				ModBus.MB_Query.Read_Quantity := 64;
				ModBus.MB_Start := TRUE;

				state:=135;
			END_IF
		END_IF
	135: (* Rispota Altri paramenti *)

		IF NOT ModBus.MB_Start  THEN

			IF ModBus.MB_MASTER.MB_Error<>0 THEN
				state := 300;
			ELSE

